	(*═════════════════════════════════════════════════════════*)
	(*  External Systems and I/O    *)
	(*═════════════════════════════════════════════════════════*)
	controlfb_control_b_start                                  , (* BOOL *)
	controlfb_control_b_stop                                   , (* BOOL *)
	controlfb_control_b_shutdown                               , (* BOOL *)
	controlfb_control_b_Reset                                  , (* BOOL *)
	controlfb_control_b_SystemShutdown                         , (* BOOL *)
	controlfb_control_b_EMstop                                 , (* BOOL *)
	controlfb_control_b_ClearHistory                           , (* BOOL *)
	controlfb_control_b_ActivateSettings                       , (* BOOL *)
	controlfb_control_b_startDeHum                             , (* BOOL *)
	controlfb_Operation_inputgrid_b_SyncClose                  , (* BOOL *)
	controlfb_Operation_Genset_b_manualStart                   , (* BOOL *)
	controlfb_Operation_PSB_b_SyncClose                        , (* BOOL *)
	controlfb_Operation_charger_b_StartCharging                , (* BOOL *)
	controlfb_Operation_charger_b_ResetCharger                 , (* BOOL *)
	controlfb_Operation_system_r_NominalVoltage                , (* REAL *)
	controlfb_Operation_system_r_NominalFrequency              , (* REAL *)
	controlfb_Operation_system_r_Pset                          , (* REAL *)
	controlfb_Operation_system_r_Qset                          , (* REAL *)
	controlfb_Operation_system_r_PFset                         , (* REAL *)
	controlfb_Operation_system_b_PFsetEnable                   , (* BOOL *)
	controlfb_Operation_system_b_SounderMute                   , (* BOOL *)
	controlfb_Operation_system_b_SounderTest                   , (* BOOL *)
	controlfb_Operation_system_b_GenGridModeTrans              , (* BOOL *)
	controlfb_Operation_system_b_GridTakeOverEnable            , (* BOOL *)
	controlfb_Operation_parallel_b_DetectSlaves                , (* BOOL *)
	controlfb_Operation_parallel_r_ActivePowerSlave1           , (* REAL *)
	controlfb_Operation_parallel_r_ReactivePowerSlave1         , (* REAL *)
	controlfb_Operation_parallel_r_ActivePowerSlave2           , (* REAL *)
	controlfb_Operation_parallel_r_ReactivePowerSlave2         , (* REAL *)
	controlfb_Operation_BMS_b_ManualStartHVDC                  , (* BOOL *)
	controlfb_SoftSettings_inputgrid_PeakshaveMode             , (* ePeakshaveMode *)
	controlfb_SoftSettings_inputgrid_setpointTimeslot1_r_SocTarget, (* REAL *)
	controlfb_SoftSettings_inputgrid_setpointTimeslot1_r_IdleChargePower, (* REAL *)
	controlfb_SoftSettings_inputgrid_setpointTimeslot1_r_FeedInCurrentLimitSoft, (* REAL *)
	controlfb_SoftSettings_inputgrid_setpointTimeslot1_r_SupplyCurrentLimitSoft, (* REAL *)
	controlfb_SoftSettings_inputgrid_setpointTimeslot2_r_SocTarget, (* REAL *)
	controlfb_SoftSettings_inputgrid_setpointTimeslot2_r_IdleChargePower, (* REAL *)
	controlfb_SoftSettings_inputgrid_setpointTimeslot2_r_FeedInCurrentLimitSoft, (* REAL *)
	controlfb_SoftSettings_inputgrid_setpointTimeslot2_r_SupplyCurrentLimitSoft, (* REAL *)
	controlfb_SoftSettings_inputgrid_b_BreakerControl          , (* BOOL *)
	controlfb_SoftSettings_inputgrid_b_ReverseCTDirection      , (* BOOL *)
	controlfb_SoftSettings_inputgrid_ui_CTrange                , (* UINT *)
	controlfb_SoftSettings_inputgrid_r_VTratio                 , (* REAL *)
	controlfb_SoftSettings_inputgrid_b_GridCodesActive         , (* BOOL *)
	controlfb_SoftSettings_inputgrid_b_WeakGridInput           , (* BOOL *)
	controlfb_SoftSettings_inputgrid_breaker_AutoConnect       , (* BOOL *)
	controlfb_SoftSettings_inputgrid_breaker_ShutdownDisconnect, (* BOOL *)
	controlfb_SoftSettings_inputgrid_breaker_EMstopDisconnect  , (* BOOL *)
	controlfb_SoftSettings_inputgrid_breaker_CurrentLimitDisconnect, (* BOOL *)
	controlfb_SoftSettings_inputgrid_breaker_CurrentLimitRetries, (* BYTE *)
	controlfb_SoftSettings_inputgenset_b_AutoStartStop         , (* BOOL *)
	controlfb_SoftSettings_inputgenset_b_HydridMode            , (* BOOL *)
	controlfb_SoftSettings_inputgenset_b_EnableSchedule        , (* BOOL *)
	controlfb_SoftSettings_inputgenset_setpointTimeslot1_r_SoCStart, (* REAL *)
	controlfb_SoftSettings_inputgenset_setpointTimeslot1_r_SoCStop, (* REAL *)
	controlfb_SoftSettings_inputgenset_setpointTimeslot1_r_BatteryloadStart, (* REAL *)
	controlfb_SoftSettings_inputgenset_setpointTimeslot1_r_BatteryloadStop, (* REAL *)
	controlfb_SoftSettings_inputgenset_setpointTimeslot1_b_StartAtBatteryError, (* BOOL *)
	controlfb_SoftSettings_inputgenset_setpointTimeslot2_r_SoCStart, (* REAL *)
	controlfb_SoftSettings_inputgenset_setpointTimeslot2_r_SoCStop, (* REAL *)
	controlfb_SoftSettings_inputgenset_setpointTimeslot2_r_BatteryloadStart, (* REAL *)
	controlfb_SoftSettings_inputgenset_setpointTimeslot2_r_BatteryloadStop, (* REAL *)
	controlfb_SoftSettings_inputgenset_setpointTimeslot2_b_StartAtBatteryError, (* BOOL *)
	controlfb_SoftSettings_inputgenset_b_PSBExtGensetMonitoring, (* BOOL *)
	controlfb_SoftSettings_inputgenset_b_FreqProtectionEnable  , (* BOOL *)
	controlfb_SoftSettings_inputgenset_Generator_e_GensetMode  , (* eGensetMode *)
	controlfb_SoftSettings_inputgenset_Generator_b_GensetLoadshareLine, (* BOOL *)
	controlfb_SoftSettings_inputgenset_Generator_r_RatedPower  , (* REAL *)
	controlfb_SoftSettings_inputgenset_Generator_r_powerloadMax, (* REAL *)
	controlfb_SoftSettings_inputgenset_Generator_r_PowerloadMin, (* REAL *)
	controlfb_SoftSettings_inputgenset_Generator_r_PowerloadEff, (* REAL *)
	controlfb_SoftSettings_inputgenset_Generator_r_ramprate    , (* REAL *)
	controlfb_SoftSettings_inputgenset_Generator_ui_CooldownTime, (* UINT *)
	controlfb_SoftSettings_inputgenset_Generator_ui_WarmupTime , (* UINT *)
	controlfb_SoftSettings_inputgenset_Loadbank_b_Enable       , (* BOOL *)
	controlfb_SoftSettings_inputgenset_Loadbank_r_PowerRating  , (* REAL *)
	controlfb_SoftSettings_inputgenset_Loadbank_r_PowerStepSize, (* REAL *)
	controlfb_SoftSettings_PSB_PeakshaveMode                   , (* ePeakshaveMode *)
	controlfb_SoftSettings_PSB_setpointTimeslot1_r_SocTarget   , (* REAL *)
	controlfb_SoftSettings_PSB_setpointTimeslot1_r_IdleChargePower, (* REAL *)
	controlfb_SoftSettings_PSB_setpointTimeslot1_r_FeedInCurrentLimitSoft, (* REAL *)
	controlfb_SoftSettings_PSB_setpointTimeslot1_r_SupplyCurrentLimitSoft, (* REAL *)
	controlfb_SoftSettings_PSB_setpointTimeslot2_r_SocTarget   , (* REAL *)
	controlfb_SoftSettings_PSB_setpointTimeslot2_r_IdleChargePower, (* REAL *)
	controlfb_SoftSettings_PSB_setpointTimeslot2_r_FeedInCurrentLimitSoft, (* REAL *)
	controlfb_SoftSettings_PSB_setpointTimeslot2_r_SupplyCurrentLimitSoft, (* REAL *)
	controlfb_SoftSettings_PSB_b_BreakerControl                , (* BOOL *)
	controlfb_SoftSettings_PSB_b_ReverseCTDirection            , (* BOOL *)
	controlfb_SoftSettings_PSB_ui_CTrange                      , (* UINT *)
	controlfb_SoftSettings_PSB_r_VTratio                       , (* REAL *)
	controlfb_SoftSettings_system_b_EnableSchedule             , (* BOOL *)
	controlfb_SoftSettings_system_b_EnableTransportMode        , (* BOOL *)
	controlfb_SoftSettings_system_b_EcoModeEnable              , (* BOOL *)
	controlfb_SoftSettings_system_e_UgridPowerMode             , (* eUgridPowerMode *)
	controlfb_SoftSettings_system_e_NetcontactorMode           , (* eNetcontMode *)
	controlfb_SoftSettings_system_e_UgridPowerLimitingMode     , (* ePLM *)
	controlfb_SoftSettings_system_b_AutomaticSwitching         , (* BOOL *)
	controlfb_SoftSettings_system_b_AMF                        , (* BOOL *)
	controlfb_SoftSettings_system_r_FrequencyDroop             , (* REAL *)
	controlfb_SoftSettings_system_r_VoltageDroop               , (* REAL *)
	controlfb_SoftSettings_system_r_SocMin                     , (* REAL *)
	controlfb_SoftSettings_system_r_SocMax                     , (* REAL *)
	controlfb_SoftSettings_system_r_PDischargeLimit            , (* REAL *)
	controlfb_SoftSettings_system_r_PChargeLimit               , (* REAL *)
	controlfb_SoftSettings_system_r_AMax                       , (* REAL *)
	controlfb_SoftSettings_system_s_SystemName                 , (* STRING(18) *)
	controlfb_SoftSettings_system_s_SMSnumber                  , (* STRING(18) *)
	controlfb_SoftSettings_system_ScheduleTimeSlot1_b_active   , (* BOOL *)
	controlfb_SoftSettings_system_ScheduleTimeSlot1_usi_DayOfWeek, (* USINT *)
	controlfb_SoftSettings_system_ScheduleTimeSlot1_usi_HourOfDay, (* USINT *)
	controlfb_SoftSettings_system_ScheduleTimeSlot1_usi_MinuteOfHour, (* USINT *)
	controlfb_SoftSettings_system_ScheduleTimeSlot2_b_active   , (* BOOL *)
	controlfb_SoftSettings_system_ScheduleTimeSlot2_usi_DayOfWeek, (* USINT *)
	controlfb_SoftSettings_system_ScheduleTimeSlot2_usi_HourOfDay, (* USINT *)
	controlfb_SoftSettings_system_ScheduleTimeSlot2_usi_MinuteOfHour, (* USINT *)
	controlfb_SoftSettings_system_by_LEDbrightness             , (* BYTE *)
	controlfb_SoftSettings_setup_e_AcInputType                 , (* eAcInputType *)
	controlfb_SoftSettings_setup_b_MasterSlaveMode             , (* BOOL *)
	controlfb_SoftSettings_setup_b_PeakshaveBoxEnable          , (* BOOL *)
	controlfb_SoftSettings_setup_e_Gridmode                    , (* eGridmode *)
	controlfb_SoftSettings_setup_e_DcCouplingType              , (* eDCinputType *)
	controlfb_SoftSettings_setup_b_ExtGenset                   , (* BOOL *)
	controlfb_HardSettings_setup_e_ControlSource               , (* eControlSources *)
	controlfb_HardSettings_charger_r_PowerMax                  , (* REAL *)
	controlfb_HardSettings_parallel_b_MasterSlaveEnabled       , (* BOOL *)
	controlfb_HardSettings_parallel_b_UnitIsMaster             , (* BOOL *)
	controlfb_HardSettings_parallel_b_ShutdownOnCommError      , (* BOOL *)
	controlfb_HardSettings_parallel_b_EffiencyMode             , (* BOOL *)
	controlfb_HardSettings_parallel_r_VoltageDroop             , (* REAL *)
	controlfb_HardSettings_parallel_r_FrequencyDroop           , (* REAL *)
	controlfb_HardSettings_system_r_PDischargeLimit            , (* REAL *)
	controlfb_HardSettings_system_r_PChargeLimit               , (* REAL *)
	controlfb_HardSettings_system_r_SMax                       , (* REAL *)
	controlfb_HardSettings_system_r_Amax                       , (* REAL *)
	controlfb_HardSettings_system_e_EarthingSystem             , (* eEarthingSystems *)
	controlfb_HardSettings_system_a_ui_InputCurrentLimit_1     , (* UINT *)
	controlfb_HardSettings_system_a_ui_InputCurrentLimit_2     , (* UINT *)
	controlfb_HardSettings_system_a_ui_OutputCurrentLimit_1    , (* UINT *)
	controlfb_HardSettings_system_a_ui_OutputCurrentLimit_2    , (* UINT *)
	controlfb_HardSettings_system_a_ui_OutputCurrentLimit_3    , (* UINT *)
	Generator_CommunicationOK                                  , (* BOOL *)
	Generator_FuelLow                                          , (* BOOL *)
	Generator_FuelCritical                                     , (* BOOL *)
	Generator_bGenBreakerClosed                                , (* BOOL *)
	Generator_bMainBreakerClosed                               , (* BOOL *)
	Generator_bGenRunning                                      , (* BOOL *)
	Generator_bGenVoltFreqOK                                   , (* BOOL *)
	Generator_bMainsFailure                                    , (* BOOL *)
	Generator_eActiveGenMode                                   , (* eGenOperationMode *)
	Generator_bIslandModeActive                                , (* BOOL *)
	Generator_bAMFActive                                       , (* BOOL *)
	Generator_bPeakshaveActive                                 , (* BOOL *)
	Generator_bFixedPowerActive                                , (* BOOL *)
	Generator_ar_LineVoltage_AVG                               , (* REAL *)
	Generator_ar_LineVoltage_L1                                , (* REAL *)
	Generator_ar_LineVoltage_L2                                , (* REAL *)
	Generator_ar_LineVoltage_L3                                , (* REAL *)
	Generator_ar_PhaseVoltage_AVG                              , (* REAL *)
	Generator_ar_PhaseVoltage_L1                               , (* REAL *)
	Generator_ar_PhaseVoltage_L2                               , (* REAL *)
	Generator_ar_PhaseVoltage_L3                               , (* REAL *)
	Generator_ar_Frequency_AVG                                 , (* REAL *)
	Generator_ar_Frequency_L1                                  , (* REAL *)
	Generator_ar_Frequency_L2                                  , (* REAL *)
	Generator_ar_Frequency_L3                                  , (* REAL *)
	Generator_ar_Current_AVG                                   , (* REAL *)
	Generator_ar_Current_L1                                    , (* REAL *)
	Generator_ar_Current_L2                                    , (* REAL *)
	Generator_ar_Current_L3                                    , (* REAL *)
	Generator_ar_PowerFactor_AVG                               , (* REAL *)
	Generator_ar_ActivePower_AVG                               , (* REAL *)
	Generator_ar_ActivePower_L1                                , (* REAL *)
	Generator_ar_ActivePower_L2                                , (* REAL *)
	Generator_ar_ActivePower_L3                                , (* REAL *)
	Generator_ar_ReactivePower_AVG                             , (* REAL *)
	Generator_ar_ApparentPower_AVG                             , (* REAL *)
	HartingIO_b_DigitalInput1Active                            , (* BOOL *)
	HartingIO_b_DigitalInput2Active                            , (* BOOL *)
	HartingIO_b_GenLowFuel                                     , (* BOOL *)
	HartingIO_b_ExtSystemShutdownRequest                       , (* BOOL *)
	HartingIO_b_ExtEMstopOK                                    , (* BOOL *)
	HartingIO_b_ExtEMstopActive                                , (* BOOL *)
	last
) DINT;
END_TYPE

// ---- POUs/MonitoringControl/IoT/DUTS/eIoTCommVersion.TcDUT
{attribute 'qualified_only'}
{attribute 'strict'}
TYPE eIoTCommVersion :
(
	V1 := 0,
	V2 := 1
);
END_TYPE

// ---- POUs/MonitoringControl/IoT/DUTS/eLogType.TcDUT
{attribute 'qualified_only'}
TYPE eLogType :
(
	none := 0,
	nuc := 1,
	cloud := 2
)UINT;
END_TYPE

// ---- POUs/MonitoringControl/IoT/DUTS/eUpdate.TcDUT
{attribute 'qualified_only'}
TYPE eUpdate :
(
	Fast			:= 0,
	Slow			:= 1,
	OnChange 		:= 2, //Updates only of variable has changed from previous value, but additionaly exactly once at system startup.
	Daily			:= 3
)UINT;
END_TYPE

// ---- POUs/MonitoringControl/IoT/DUTS/e_ORAttributeType.TcDUT
{attribute 'qualified_only'}
{attribute 'strict'}
TYPE e_ORAttributeType :
(
	text := 0,
	number := 2,
	integer := 3,
	JSON := 4
);
END_TYPE

// ---- POUs/MonitoringControl/IoT/DUTS/ST_AutoProvisioning.TcDUT
TYPE ST_AutoProvisioning :
	STRUCT
		sType	: STRING;
		sRealm	: STRING;
		sError	: STRING;
	END_STRUCT
END_TYPE

// ---- POUs/MonitoringControl/IoT/DUTS/ST_IotProps.TcDUT
TYPE ST_IotProps :
STRUCT
	sName		: STRING;
	sValue		: STRING(2000);
	eUpdate 	: eUpdate;
	st_RW		: ST_RW;
	pAdress		: PVOID;
	diSize		: DINT;
	ClassType : __SYSTEM.TYPE_CLASS;
	bNumber		: BOOL;
	bJson		: BOOL;
END_STRUCT
END_TYPE

// ---- POUs/MonitoringControl/IoT/DUTS/ST_RW.TcDUT
TYPE ST_RW :
STRUCT
	ReadFromNUC : BOOL:= FALSE;//enabling Read and Write can create unintended behaviour, consider feedback var
	WriteToNUC: BOOL:=FALSE ; //enabling Read and Write can create unintended behaviour, consider feedback var
END_STRUCT
END_TYPE

// ---- POUs/MonitoringControl/IoT/DUTS/ST_Supervisor.TcDUT
TYPE ST_Supervisor :
	STRUCT
		DATA	: STRING;
		ERROR	: STRING;
	END_STRUCT
END_TYPE

// ---- POUs/MonitoringControl/IoT/DUTS/ST_VarBuffer.TcDUT
TYPE ST_VarBuffer :
STRUCT
	sValue 	  : STRING(2000);
	pAdress   : PVOID;
	diSize	  : DINT;  
	ClassType : __SYSTEM.TYPE_CLASS;
	bNumber   : BOOL;
END_STRUCT
END_TYPE

// ---- POUs/MonitoringControl/IoT/_Structs/ST_IoTDataHMI.TcDUT
TYPE ST_IoTDataHMI :
STRUCT
	Label 				: STRING;
	Varname				: eDataMappingVarNames;
	Unit				: STRING(20);
	LogType 			: eLogType; 
	LogInterval 		: eUpdate;
	b_IOTWriteAllowed	: BOOL;
END_STRUCT
END_TYPE

// ---- POUs/MonitoringControl/IoT/_Structs/ST_IotData_credits.TcDUT
TYPE ST_IotData_credits :
STRUCT
	TotalCredits 		: DINT := 100;
	RemainingCredits	: DINT;
	UsedCredits			: DINT;
END_STRUCT
END_TYPE

// ---- POUs/MonitoringControl/IoT/_Structs/st_IOT_params.TcDUT
TYPE st_IOT_params :
STRUCT
	b_controlEnable			: 	BOOL := FALSE;
	r_UpdateTimeFast		: 	REAL := 15; //seconds
	r_UpdateTimeSlow		: 	REAL := 60; //seconds
	IotCommVersion			: 	eIotCommVersion;
	DefaultLoggingBudget	:	UINT	:= 100;
END_STRUCT
END_TYPE

// ---- POUs/MonitoringControl/IoT/_Structs/ST_IOT_SentStateLog.TcDUT
TYPE ST_IOT_SentStateLog :
STRUCT
	bUpdate			: BOOL;
	bMessageSent	: BOOL;
	LastIndexSent	: INT;
	LastIndex		: INT;
END_STRUCT
END_TYPE

// ---- POUs/MonitoringControl/ProfinetController/enums/eExternalControlMode.TcDUT
{attribute 'qualified_only'}
{attribute 'strict'}
TYPE eExternalControlMode :
(
	off := 0,
	Readonly := 1,
	BasicControl := 2,
	AdvancedControl := 3
);
END_TYPE

// ---- POUs/MonitoringControl/ProfinetController/enums/GenGridMode.TcDUT
{attribute 'qualified_only'}
{attribute 'strict'}
TYPE GenGridMode :
(
	none := 0,
	Grid := 1,
	GridDisconnected := 11,
	GridToNone := 12,
	Genset := 2
);
END_TYPE

// ---- POUs/MonitoringControl/ProfinetController/enums/uSWversion.TcDUT
TYPE uSWversion :
UNION
	a4byte_SWVer 	: 	ARRAY[0..3] OF BYTE;
	UD_SWVer		:	UDINT; 
END_UNION
END_TYPE

// ---- POUs/MonitoringControl/ProfinetController/Structs/future use/ST_PNInput_DCBusExpansion.TcDUT
TYPE ST_PNInput_DCBusExpansion :
STRUCT
	ControlBits	:	DWORD;
END_STRUCT
END_TYPE

// ---- POUs/MonitoringControl/ProfinetController/Structs/future use/ST_PNInput_DCCharger.TcDUT
TYPE ST_PNInput_DCCharger :
STRUCT
	Controlbits	:	DWORD;
	//b_enable?
	//b_resetCharger
	//b_StartCharging
	Powerlimit	:	DWORD;
END_STRUCT
END_TYPE

// ---- POUs/MonitoringControl/ProfinetController/Structs/future use/ST_PNInput_ParallelOperation.TcDUT
TYPE ST_PNInput_ParallelOperation :
STRUCT
	Controlbits			:	DWORD;
	//b_DetectSlaves	
	r_ActivePower		:	DWORD;
	r_reactivePower		:	DWORD;
END_STRUCT
END_TYPE

// ---- POUs/MonitoringControl/ProfinetController/Structs/future use/ST_PNOutput_DCCharger.TcDUT
TYPE ST_PNOutput_DCCharger :
STRUCT
	statusbits		:	DWORD;
	ChargerStatus	:	DWORD;
	ChargePower		:	DWORD;
END_STRUCT
END_TYPE

// ---- POUs/MonitoringControl/ProfinetController/Structs/future use/ST_PNOutput_DCExpansion.TcDUT
TYPE ST_PNOutput_DCExpansion :
STRUCT
	statusbits	: DWORD;
	Busvoltage	: DWORD;
	RatedPower	: DWORD;
	LoadPercentage	: DWORD;
	CurrentPower	: DWORD;
END_STRUCT
END_TYPE

// ---- POUs/MonitoringControl/ProfinetController/Structs/future use/ST_PNOutput_ParallelOperation.TcDUT
TYPE ST_PNOutput_ParallelOperation :
STRUCT
	statusbits		:	DWORD;
	ActivePower		:	DWORD;
	ReactivePower	:	DWORD;
END_STRUCT
END_TYPE

// ---- POUs/MonitoringControl/ProfinetController/Structs/NestedStructs/ST_PNInput_ACDCCharger.TcDUT
TYPE ST_PNInput_ACDCCharger :
STRUCT
	w_Control			:	WORD;
	ui_ACCurrentlimit	:	UINT	:=	0;
	UI_Pset				:	UINT	:=	0;
	ui_SocMaxLimit		:	UINT	:=	100;
	ui_MinGridVoltage	:	Uint	:=	360;
END_STRUCT
END_TYPE

// ---- POUs/MonitoringControl/ProfinetController/Structs/NestedStructs/ST_PNInput_Battery.TcDUT
TYPE ST_PNInput_Battery :
STRUCT
	w_Control		:	WORD;
	ui_SocMinLimit	:	UINT	:=	0;
	ui_SocMaxLimit	:	UINT	:=	100;
END_STRUCT
END_TYPE

// ---- POUs/MonitoringControl/ProfinetController/Structs/NestedStructs/ST_PNInput_GenControl.TcDUT
TYPE ST_PNInput_GenControl :
STRUCT
	w_Control			:	WORD;
	ui_SOCStart			:	UINT;
	ui_SOCStop			:	UINT;
	ui_BattLoadStart	:	UINT;
	ui_BattLoadStop		:	UINT;
	ui_GenPowerMode		:	UINT;
	ui_GenRatedPower	:	UINT;
	ui_GenMaxPowerLevel	:	UINT;
	ui_GenEffPowerLevel	:	UINT;
	ui_GenMinPowerLevel	:	UINT;
	ui_GenWarmupTime	:	UINT;
	ui_GenCooldownTime	:	UINT;
	ui_IsoPowerRamp		:	UINT;
	ui_GeneratorSetpoint : 	UINT;
	ui_StartStopControl	:	uint;	
END_STRUCT
END_TYPE

// ---- POUs/MonitoringControl/ProfinetController/Structs/NestedStructs/ST_PNInput_General.TcDUT
TYPE ST_PNInput_General :
STRUCT
	W_Control				:	WORD;
	ui_HeatBeat				:	UINT;
	ui_GridMode				:	UINT;
	ui_GridFormingSubMode	:	UINT;	
	ui_Earthingsystem		:	UINT;
	GridConnectionMode		:	UINT;
	PrimaryDigOutState		:	UINT := 99;
	SecondaryDigOutState	:	UINT := 99;
	PrimaryDigInState		:	UINT := 99;
	SecondaryDiginState		:	UINT := 99;
END_STRUCT
END_TYPE

// ---- POUs/MonitoringControl/ProfinetController/Structs/NestedStructs/ST_PNInput_InputField.TcDUT
TYPE ST_PNInput_InputField :
STRUCT
	w_Control				:	WORD;
	InputConnectionType		:	UINT;
//	ui_FeedInCurrentLimit	:	UINT;
//	ui_FeedOutCurrentLimit	:	UINT;
//	ui_IdleChargePower 		:	UINT;
//	ui_SocTarget			:	UINT;
//	ui_InputConnectionType	:	UINT;
END_STRUCT                       
END_TYPE

// ---- POUs/MonitoringControl/ProfinetController/Structs/NestedStructs/ST_PNInput_InputGridControl.TcDUT
TYPE ST_PNInput_InputGridControl :
STRUCT
	w_Control				:	WORD;
	ui_FeedInCurrentLimit	:	UINT;
	ui_SupplyCurrentLimit	:	UINT;
	ui_CurrentLimitRetries	:	UINT;
	ui_ContactorControl		:	uint;
END_STRUCT
END_TYPE

// ---- POUs/MonitoringControl/ProfinetController/Structs/NestedStructs/ST_PNInput_PeakShaveBox.TcDUT
TYPE ST_PNInput_PeakShaveBox :
STRUCT
	w_Control			:	WORD;
	ui_FeedInCurrentLimit	:	UINT;
	ui_SupplyCurrentLimit	:	UINT;
	ui_VTRatio				:	UINT;
	UI_CTRatio				:	UINT;
END_STRUCT
END_TYPE

// ---- POUs/MonitoringControl/ProfinetController/Structs/NestedStructs/ST_PNInput_Powerstack.TcDUT
TYPE ST_PNInput_Powerstack :
STRUCT
	w_Control			:	WORD;
	ui_NominalVoltage	:	UINT;
	ui_NominalFrequency	:	UINT;
	i_Pset				:	INT;
	i_Qset				:	INT;
	i_PFset				:	INT;
	ui_FrequencyDroop	:	UINT;
	ui_VoltageDroop		:	UINT;
	ui_PowerRampRate	:	UINT;
	ui_SOCDroopUpshiftStart		:	UINT;
	ui_SOCDroopDownShiftStart	:	UINT;
	ui_PowerLimitMode	:	UINT;
	ui_ACCurrentLimit	:	UINT;
END_STRUCT
END_TYPE

// ---- POUs/MonitoringControl/ProfinetController/Structs/NestedStructs/ST_PNOutput_ACDCCharger.TcDUT
TYPE ST_PNOutput_ACDCCharger :
STRUCT
	w_Status						: WORD;
	w_Warnings						: WORD;
	w_Faults						: WORD;
	ui_ChargerStatus				: WORD;
	TotalChargerPower				: WORD;
	AvailableChargePower			: UINT;
	ActivePower						: UINT;
	Frequency						: UINT;
	VoltageAB						: UINT;
	VoltageBC						: UINT;
	VoltageCA						: UINT;
	CurrentL1						: UINT;
	CurrentL2						: UINT;
	CurrentL3						: UINT;
	ui_ACCurrentLimitAct			: UINT;
	ui_PSetAct						: UINT;
	ui_SocLimitAct					: UINT;
	ui_MinGridVoltageAct			: UINT;
END_STRUCT
END_TYPE

// ---- POUs/MonitoringControl/ProfinetController/Structs/NestedStructs/ST_PNOutput_Battery.TcDUT
TYPE ST_PNOutput_Battery :
STRUCT
	ui_Status						: UINT;
	w_Warnings						: WORD;
	w_Faults						: WORD;

	ui_SOC							: UINT;
	ui_SOH							: UINT;
	ui_DClinkVoltage 				: UINT;
	i_DClinkCurrent 				: INT;
	ui_MaxAllowedDischargeCurrent 	: UINT;
	ui_MaxAllowedChargeCurrent 		: UINT;
	i_MinCellTemperature 			: INT;
	i_MaxCellTemperature			: INT;
	ui_RemainingChargeEnergy 		: UINT;
	ui_RemainingDischargeEnergy 	: UINT;
	ui_CycleCount					: UINT;
END_STRUCT
END_TYPE

// ---- POUs/MonitoringControl/ProfinetController/Structs/NestedStructs/ST_PNOutput_GenControl.TcDUT
TYPE ST_PNOutput_GenControl :
STRUCT
	w_Status					:	WORD;
	w_Warnings					:	WORD;
	w_Faults					:	WORD;
	ui_GeneratorStatus			:	UINT;	
END_STRUCT
END_TYPE

// ---- POUs/MonitoringControl/ProfinetController/Structs/NestedStructs/ST_PNOutput_General.TcDUT
TYPE ST_PNOutput_General :
STRUCT
	ui_SystemState				:	UINT;
	w_SystemStatus				:	WORD;	
	w_SystemWarnings			:	WORD;
	w_SystemFaults				:	WORD;
	w_CoolingSystemStatus		:	WORD;
	w_CoolingSystemWarnings		:	WORD;
	w_CoolingSystemFaults		:	WORD;
	w_InternalSupplyStatus		:	WORD;
	w_InternalSupplyWarnings	:	WORD;
	w_InternalSupplyFaults		:	WORD;	
	ui_HeartBeatOut				:	UINT;
	ui_Gridmode					: 	UINT;
	ui_GridFormingSubMode		: 	UINT;
	udi_SerialNumber			:	UDINT;
	dw_SWVersion				:	DWORD;
	//ui_InputConnectionType		:	UINT;
END_STRUCT
END_TYPE

// ---- POUs/MonitoringControl/ProfinetController/Structs/NestedStructs/ST_PNOutput_InputField.TcDUT
TYPE ST_PNOutput_InputField:
STRUCT
	w_Status					:	WORD;
	w_Warnings					:	WORD;
	w_Faults					:	WORD;
	ui_InputConnectionType		:	UINT;
	ui_InputConnectionState		:	UINT;
	i_ActivePower				:	INT;
	i_ReactivePower				:	INT;
	i_PowerFactor				:	INT;
	ui_Frequency				:	UINT;
	ui_VoltageL1N				:	UINT;
	ui_VoltageL2N				:	UINT;
	ui_VoltageL3N				:	UINT;
	ui_VoltageL1L2				:	UINT;
	ui_VoltageL2L3				:	UINT;
	ui_VoltageL3L1				:	UINT;
	ui_CurrentL1				:	UINT;
	ui_CurrentL2				:	UINT;
	ui_CurrentL3				:	UINT;
	ui_CurrentN					:	UINT;
	ui_CurrentLimitField		:	UINT;
	udi_TotalEnergySupplied 	:	UDINT;
	udi_TotalEnergyConsumed 	:	UDINT;
	ui_Current1L1				:	UINT;
	ui_Current1L2				:	UINT;
	ui_Current1L3				:	UINT;
	ui_Current1N				:	UINT;
	ui_Current2L1				:	UINT;
	ui_Current2L2				:	UINT;
	ui_Current2L3				:	UINT;
	ui_Current2N				:	UINT;
END_STRUCT
END_TYPE

// ---- POUs/MonitoringControl/ProfinetController/Structs/NestedStructs/ST_PNOutput_InputGridControl.TcDUT
TYPE ST_PNOutput_InputGridControl :
STRUCT
	w_Status					:	WORD;
	w_Warnings					:	WORD;
	w_Faults					:	WORD;
	ui_InputGridStatus			:	UINT;
END_STRUCT
END_TYPE

// ---- POUs/MonitoringControl/ProfinetController/Structs/NestedStructs/ST_PNOutput_OutputField.TcDUT
TYPE ST_PNOutput_OutputField:
STRUCT
	w_Status					:	WORD;
	w_Warnings					:	WORD;
	w_Faults					:	WORD;
	i_ActivePower				:	INT;
	i_ReactivePower				:	INT;
	i_PowerFactor				:	INT;
	ui_Frequency				:	UINT;
	ui_VoltageL1N				:	UINT;
	ui_VoltageL2N				:	UINT;
	ui_VoltageL3N				:	UINT;
	ui_VoltageL1L2				:	UINT;
	ui_VoltageL2L3				:	UINT;
	ui_VoltageL3L1				:	UINT;
	ui_CurrentL1				:	UINT;
	ui_CurrentL2				:	UINT;
	ui_CurrentL3				:	UINT;
	ui_CurrentN					:	UINT;
	ui_CurrentLimitField		:	UINT;
	udi_TotalEnergySupplied 	:	UDINT;
	udi_TotalEnergyConsumed 	:	UDINT;
	ui_Current1L1				:	UINT;
	ui_Current1L2				:	UINT;
	ui_Current1L3				:	UINT;
	ui_Current1N				:	UINT;
	ui_Current2L1				:	UINT;
	ui_Current2L2				:	UINT;
	ui_Current2L3				:	UINT;
	ui_Current2N				:	UINT;
	ui_Current3L1				:	UINT;
	ui_Current3L2				:	UINT;
	ui_Current3L3				:	UINT;
	ui_Current3N				:	UINT;
END_STRUCT
END_TYPE

// ---- POUs/MonitoringControl/ProfinetController/Structs/NestedStructs/ST_PNOutput_PeakShaveBox.TcDUT
TYPE ST_PNOutput_PeakShaveBox:
STRUCT
	w_Status					:	WORD;
	w_Warnings					:	WORD;
	w_Faults					:	WORD;
	i_ActivePower				:	INT;
	i_ReactivePower				:	INT;
	i_PowerFactor				:	INT;
	ui_Frequency				:	UINT;
	ui_VoltageL1N				:	UINT;
	ui_VoltageL2N				:	UINT;
	ui_VoltageL3N				:	UINT;
	ui_VoltageL1L2				:	UINT;
	ui_VoltageL2L3				:	UINT;
	ui_VoltageL3L1				:	UINT;
	ui_CurrentL1				:	UINT;
	ui_CurrentL2				:	UINT;
	ui_CurrentL3				:	UINT;
	ui_CurrentN					:	UINT;
END_STRUCT
END_TYPE

// ---- POUs/MonitoringControl/ProfinetController/Structs/NestedStructs/ST_PNOutput_PowerStack.TcDUT
TYPE ST_PNOutput_PowerStack :
STRUCT
	w_Status					:	WORD;
	w_Warnings					:	WORD;
	w_Faults					:	WORD;
	
	ui_PowerStackStatus			: UINT;
	i_ActivePower				: INT;
	i_ReactivePower				: INT;
	ui_SupplyVoltage			: UINT;
	ui_Supplyfrequency			: UINT;
	ui_ACCurrent				: UINT;
	i_PsetAct					: INT;
	i_QsetAct					: INT;
	i_PFSetAct					: UINT;
	ui_LoadPercentage			: UINT;
	ui_RatedCurrent				: UINT;
	ui_RatedPower				: UINT;
	ui_DischargePowerLimit		: UINT;
	ui_ChargePowerLimit			: UINT;
	ui_ACcurrentLimit			: UINT;
	ui_ApparentPowerLimit		: UINT;
	ui_ReactivePowerLimit		: UINT;
END_STRUCT
END_TYPE

// ---- POUs/MonitoringControl/ProfinetController/Structs/NestedStructs/ST_PNOutput_ZPT.TcDUT
TYPE ST_PNOutput_ZPT :
STRUCT
	w_Status					:	WORD;
	w_Warnings					:	WORD;
	w_Errors					:	WORD;
	ui_RatedPower				:	UINT;
	ui_Powerload				:	UINT;
	i_TransformerTemperature	:	INT;
END_STRUCT
END_TYPE

// ---- POUs/MonitoringControl/ProfinetController/Structs/ST_PNcontroller_params.TcDUT
TYPE ST_PNcontroller_params :
STRUCT
	b_BigEndian				: BOOL;
	b_testComm				: BOOL;
	b_MonitoringEnable		: BOOL := TRUE;
	b_ControlEnable			: BOOL := TRUE;
	w_CommTimeOut			: WORD := 10000; // milli seconds
	TestVars				: ST_PNTest;
	Limits					: ST_ExtController_limits;
END_STRUCT
END_TYPE

// ---- POUs/MonitoringControl/ProfinetController/Structs/ST_PNinput.TcDUT
TYPE ST_PNinput :
STRUCT
	PNIOBoxState		:	WORD;
	PNIOBoxDiag			:	WORD;	
	General 			: ST_PNInput_General;
	Battery				: ST_PNInput_Battery;
	Inputfield			: ST_PNInput_InputField;
	PSB					: ST_PNInput_PeakshaveBox;
	Powerstack			: ST_PNInput_Powerstack;
	GenControl 			: ST_PNInput_GenControl;
	InputGridControl	: ST_PNInput_InputGridControl;	
	ACDCCharger			: ST_PNInput_ACDCCharger;
END_STRUCT
END_TYPE

// ---- POUs/MonitoringControl/ProfinetController/Structs/ST_PNOutput.TcDUT
TYPE ST_PNOutput :
STRUCT
	General 		: ST_PNOutput_General;
	Battery			: ST_PNOutput_Battery;
	OutputField		: ST_PNOutput_Outputfield;
	InputField		: ST_PNOutput_Inputfield;
	Powerstack 		: ST_PNOutput_Powerstack;
	PSB 			: ST_PNOutput_PeakshaveBox;
	ZPT				: ST_PNOutput_ZPT;
	GenControl 		: ST_PNOutput_GenControl;
	InputGridControl: ST_PNOutput_InputGridControl;
	ACDCCharger		: ST_PNOutput_ACDCCharger;
END_STRUCT
END_TYPE

// ---- POUs/MonitoringControl/ProfinetController/Structs/ST_PNTest.TcDUT
TYPE ST_PNTest :
STRUCT
	b_CheckMonitoring	: BOOL;
	b_MonitoringOK		: BOOL;
	s_MonitoringErr		: STRING;
	i_Pset				: INT;
	i_Qset				: INT;
	w_SetAddress		: WORD;
	w_SetValue			: WORD;
	bit_start			: BOOL;
	bit_stop			: BOOL;
	bit_Shutdown		: BOOL;
	bit_SystemShutdown	: BOOL;
	bit_Reset			: BOOL;
	bit_EMStop			: BOOL;
	bit_AdvancedControl	: BOOL;
	bit_AutoSwitching	: BOOL;
	bit_Transportmode	: BOOL;
END_STRUCT
END_TYPE

// ---- POUs/MonitoringControl/_Enums/eAcInputType.TcDUT
{attribute 'qualified_only'}
{attribute 'strict'}
TYPE eAcInputType :
(
	None 	:= 0,
	Grid 	:= 1,
	Genset	:= 2
);
END_TYPE

// ---- POUs/MonitoringControl/_Enums/eCapTestSTate.TcDUT
{attribute 'qualified_only'}
{attribute 'strict'}
TYPE eCapTestSTate :
(
	init 				:= 	0,
	WriteSerial			:=	1,
	WriteNameplateCap	:=	2,
	WriteDatetime		:=	3,
	StartSystem 		:= 	4,
	InitialCharge 		:= 	5,
	RestPeriod1			:= 	6,
	DischargeCycle 		:= 	7,
	RestPeriod2 		:= 	8,
	ChargeCycle 		:= 	9,
	RestPeriod3 		:= 	10,
	StopSystem  		:= 	11,
	done				:=	12
);
END_TYPE

// ---- POUs/MonitoringControl/_Enums/eControlSources.TcDUT
{attribute 'qualified_only'}
{attribute 'strict'}
{attribute 'to_string'}
TYPE eControlSources :
(
	Local 				:= 0,
	ExternalController 	:= 1,
	PowerNet			:= 2	
);
END_TYPE

// ---- POUs/MonitoringControl/_Enums/eDcInputType.TcDUT
{attribute 'qualified_only'}
{attribute 'strict'}
TYPE eDcInputType :
(
	None := 0,
	Dc_charger := 1, 
	Dc_extender := 2
);
END_TYPE

// ---- POUs/MonitoringControl/_Enums/eEarthingSystems.TcDUT
{attribute 'qualified_only'}
{attribute 'strict'}
TYPE eEarthingSystems :
(
	None 		:= 0,	
	TN			:= 1,
	TN_ext		:= 2,
	IT			:= 3		
);
END_TYPE

// ---- POUs/MonitoringControl/_Enums/eGridFormingMode.TcDUT
{attribute 'qualified_only'}
{attribute 'strict'}
TYPE eGridFormingMode:
(
	Island := 0,
	Droop := 1
);
END_TYPE

// ---- POUs/MonitoringControl/_Enums/eGridMode.TcDUT
{attribute 'qualified_only'}
{attribute 'strict'}
{attribute 'to_string'}
TYPE eGridMode :
(
	auto := 0,
	following := 1,
	forming	:= 2
);
END_TYPE

// ---- POUs/MonitoringControl/_Enums/eNetContactorDirection.TcDUT
{attribute 'qualified_only'}
{attribute 'strict'}
TYPE eNetContactorDirection :
(
	Left 	:= -1,
	None 	:= 0,
	Right 	:= 1
);
END_TYPE

// ---- POUs/MonitoringControl/_Enums/eOperationMode.TcDUT
{attribute 'qualified_only'}
{attribute 'strict'}
TYPE eOperationMode :
(
	Auto := 0,
	Gridfollowing := 1,
	GridForming	:= 2
);
END_TYPE

// ---- POUs/MonitoringControl/_Enums/ePeakshaveMode.TcDUT
{attribute 'qualified_only'}
{attribute 'strict'}
TYPE ePeakshaveMode :
(
	Multiphase := 0,
	Singlephase := 1
);
END_TYPE

// ---- POUs/MonitoringControl/_Enums/eSchedulerMode.TcDUT
{attribute 'qualified_only'}
{attribute 'strict'}
TYPE eSchedulerMode :
(
	continous := 0,
	daily := 1,
	weekly := 2
);
END_TYPE

// ---- POUs/MonitoringControl/_Enums/ePowerControlType.TcDUT
{attribute 'qualified_only'}
{attribute 'strict'}
{attribue 'to_string}
TYPE ePowerControlType :
(
	Current := 0,
	Power	:=1,
	Both	:= 2
);
END_TYPE

// ---- POUs/MonitoringControl/_Enums/eSystemState.TcDUT
{attribute 'qualified_only'}
{attribute 'strict'}
{attribute 'to_string'}
TYPE eSystemState :
(
	Off 			:= 0,
	Shutdown 		:= 1,
	StandBy 		:= 2,
	Conditioning 	:= 3,
	Starting		:= 4,
	Running			:= 5,
	Charging_Only	:= 6,
	Discharging_Only:= 7,
	Stopped			:= 8,
	EMstop			:= 9,
	Reset			:= 10,
	Init			:= 11,
	Transport		:= 12,
	Dehumidifying	:= 13
);
END_TYPE

// ---- POUs/MonitoringControl/_Enums/eUgridPowerMode.TcDUT
{attribute 'qualified_only'}
{attribute 'strict'}
{attribute 'to_string'}
TYPE eUgridPowerMode :
(
	auto 			:= 0,
	DroopZeroStart	:= 1,
	Droop			:= 2,
	Isochronous		:= 3,
	None			:= 4
);
END_TYPE

// ---- POUs/MonitoringControl/_Structs/ST_ExtController_Events.TcDUT
TYPE ST_ExtController_Events :
STRUCT
	b_HeartbeatFault			: BIT;
	b_couplerError				:	bit;
	
	// control limit warnings
	b_FeedInLimitOutOfRange		: BIT;
	b_SupplyLimitOutOfRange 	: BIT;
	b_IdleChargePowerOutofRange	: BIT;
	b_BatOloadStartOutOfRange	: BIT;
	b_BatOloadStopOutOfRange	: BIT;
	b_SocTargetOutOfRange		: BIT;
	b_SocStartOutOfRange		: BIT;
	b_SocStopOutOfRange			: BIT;
	b_PsetOutOfRange			: BIT;
	b_QsetOutOfRange			: BIT;
	b_PFsetOutOfRange			: BIT;
	b_NominalVoltageOutOfRange	: BIT;
	b_NominalFreqOutOfRange		: BIT;
	b_FreqDroopOutOfRange		: BIT;
	b_VoltageDroopOutOfRange	: BIT;
	b_PmaxOutOfRange			: BIT;
	b_PminOutOfRange			: BIT;
	b_SmaxOutOfRange			: BIT;
	b_AmaxOutOfRange			: BIT;
	b_PowerRamprateOutOfRange	: BIT;
	b_PSBFeedInLimitOutOfRange	: BIT;
	b_PSBSupplyLimitOutOfRange: BIT;
	b_PSBIdleChargePowerOutOfRange: BIT;
	b_PSBSoCTargetOutOfRange	: BIT;
	b_SoCHighLimitOutOfRange	: BIT;
	b_SoCLowLimitOutOfRange		: BIT;
	b_GridModeValueOutOfRange	: BIT;
	b_PowermodeValueOutOfRange	: BIT;

END_STRUCT
END_TYPE

// ---- POUs/MonitoringControl/_Structs/ST_ExtController_get.TcDUT
TYPE ST_ExtController_get :
STRUCT
	control							: ST_ControlVars;
	Operation						: ST_OperationVars;
	SoftSettings					: ST_SoftSettings;
	HardSettings					: ST_HardSettings;
	events							: ST_ExtController_Events;
	b_AdvancedControl				: BOOL;
	ui_Heartbeat					: UINT;
	s_dashboardID					: STRING;
	b_Active						: BOOL;
	e_ConnectionState				: eConnectionState;
	s_OutputJson					: STRING(2000);
	LoggingBudgetOK					: BOOL := TRUE;
END_STRUCT
END_TYPE

// ---- POUs/MonitoringControl/_Structs/ST_ExtController_limits.TcDUT
TYPE ST_ExtController_limits :
STRUCT
	r_InputCtLimit			: REAL := 800;
	r_InverterPowerLimit	: REAL := 360;
	r_InverterCurrentLimit	: REAL := 520;
	r_NominalVoltageMin		: REAL := 360;
	r_NominalVoltageMax		: REAL := 440;
	r_NominalFreqMin		: REAL := 47.5;
	r_NominalFreqMax		: REAL := 52.5;
	r_DroopMax				: REAL := 10; 
	r_PowerRampLimit		: REAL := 300; //%/s
	r_PSBCtLimit			: REAL := 4000;
END_STRUCT
END_TYPE

// ---- POUs/MonitoringControl/_Structs/ST_ExtController_Set.TcDUT
TYPE ST_ExtController_Set :
STRUCT
	b_available				: BOOL;
END_STRUCT
END_TYPE

// ---- POUs/MonitoringControl/_Structs/ST_PLCPersistentVars.TcDUT
TYPE ST_PLCPersistentVars :
STRUCT
	Hardsettings					: ST_HardSettings; 
	Softsettings					: ST_Softsettings;
END_STRUCT
END_TYPE

// ---- POUs/Objects/4Grouter/Struct/dwtoreal.TcDUT
TYPE dwtoreal :
UNION
	Registers	:	ARRAY[1..2] OF WORD;
	dwordvalue	:	dword;
	realvalue	:	REAL;
END_UNION
END_TYPE

// ---- POUs/Objects/4Grouter/Struct/eModemState.TcDUT
{attribute 'qualified_only'}
//{attribute 'strict'}
TYPE eModemState :
(
	Disconnected := 0,
	Connected := 1
);
END_TYPE

// ---- POUs/Objects/4Grouter/Struct/eNetworkState.TcDUT
{attribute 'qualified_only'}
//{attribute 'strict'}
TYPE eNetworkState :
(
	unknown := 0,
	searching := 1,
	Unregistered := 2,
	Registered := 3,
	Roaming := 4
	);
END_TYPE

// ---- POUs/Objects/4Grouter/Struct/eSimSelectionMode.TcDUT
{attribute 'qualified_only'}
{attribute 'strict'}
TYPE eSimSelectionMode :
(
	auto := 0,
	force_sim1 := 1,
	force_sim2 := 2
);
END_TYPE

// ---- POUs/Objects/4Grouter/Struct/eSimState.TcDUT
{attribute 'qualified_only'}
//{attribute 'strict'}
TYPE eSimState :
(
	no_sim := 0,
	Inserted := 1,
	active := 2,
	pin_fault := 3
);
END_TYPE

// ---- POUs/Objects/4Grouter/Struct/eSMSStatus.TcDUT
{attribute 'qualified_only'}
//{attribute 'strict'}
TYPE eSMSStatus :
(
	Idle 			:= 	0,
	NewMessage 		:= 	1,
	SendingMessage 	:= 	2,
	error			:=	3
);
END_TYPE

// ---- POUs/Objects/4Grouter/Struct/eWifiSecurityTypes.TcDUT
{attribute 'qualified_only'}
{attribute 'strict'}
{attribute 'to_string'}
TYPE eWifiSecurityTypes :
(
	none := 0,
	PSK2 := 1,
	SAE  := 2,
	SAE_mixed := 3,
	PSK := 4	
);
END_TYPE

// ---- POUs/Objects/4Grouter/Struct/eWifiStatus.TcDUT
{attribute 'qualified_only'}
TYPE eWifiStatus :
(
	invalid := 0,
	off := 1,
	searching := 2,
	Connected := 3,
	Starting := 4,
	Active := 5
);
END_TYPE

// ---- POUs/Objects/4Grouter/Struct/st_Device.TcDUT
TYPE st_Device :
STRUCT
	SystemUptime	:	UDINT;	
	Temperature		:	REAL;
	RouterSerial	:	STRING(32);
END_STRUCT
END_TYPE

// ---- POUs/Objects/4Grouter/Struct/st_GPS.TcDUT
TYPE st_GPS :
STRUCT
	Latitude 	: 	REAL;
	Longitude 	: 	REAL;
	FixTime 	: 	STRING(32);
	DateTime	:	DT;
	Speed		:	REAL;
	SatCount	:	UINT;
	Accuracy	:	REAL;	
END_STRUCT
END_TYPE

// ---- POUs/Objects/4Grouter/Struct/st_mobile.TcDUT
TYPE st_mobile :
STRUCT
	NetworkOperator				:	STRING(32);
	NetworkInfo					:	STRING(32);
	NetworkType					:	STRING(32);
	RSSI						:	DINT;
	ui_Sim1DataSendMonth		:	UINT;
	ui_Sim1DataReceivedMonth	:	UINT;
	ui_Sim2DataSendMonth		:	UINT;
	ui_Sim2DataReceivedMonth	:	UINT;
	s_EmergencySMSNumber		:	STRING(20);
	s_SecondarySMSNumber		:	STRING(20);
	s_EmergencySMSDevName		:	STRING(18);
	st_LatestSMSMessage			:	STRING(80);
	ModemState					:	eModemState;
	NetworkState				:	eNetworkState;
	ui_ActiveSim				:	UINT;
	SimStatus					:	eSimState;
END_STRUCT
END_TYPE

// ---- POUs/Objects/4Grouter/Struct/st_router_get.TcDUT
TYPE st_router_get :
STRUCT
	Device 		: 	st_Device;
	GPS			:	st_GPS;
	Mobile		:	st_mobile;
	Wifi		:	st_Wifi;
	e_SMSStatus : 	eSMSStatus;
	Events		:	st_Router_Events;
END_STRUCT
END_TYPE

// ---- POUs/Objects/4Grouter/Struct/ST_Router_params.TcDUT
TYPE ST_Router_params :
STRUCT
	IP_TELTONIKA		: STRING(16) := '192.168.1.1';
	MBPort_TELTONIKA 	: UINT := 502;
	T_MBTimeout			: TIME := T#2S;
	MinimumPhoneNumberLength	:UINT := 10;
	
	//temporary setup via stparams until integrated into HMI
	ManualSettings		:	st_router_set;
END_STRUCT
END_TYPE

// ---- POUs/Objects/4Grouter/Struct/st_Router_Events.TcDUT
TYPE st_Router_Events :
STRUCT
	b_MBCommWarning		:	BOOL;
	b_NoSimWarning		:	BOOL;
	b_NoNetworkWarning	: 	BOOL;
	b_noGPSFixWarning	:	BOOL;
	b_SMSNotSendError	:	BOOL; 
	b_NoSMSNumberAvailable	:	BOOL;
	b_TimeUpdateFailed 	: BOOL;
END_STRUCT
END_TYPE

// ---- POUs/Objects/4Grouter/Struct/ST_Router_set.TcDUT
TYPE ST_Router_set :
STRUCT
	EnableWifiClient	:	BOOL;
	WifiClientSSID		:	STRING(32) := 'MachineAccessPoint@VDL';
	WifiClientPass		:	STRING(32) := 'e4ff1c12kLL';
	WifiClientSecType	:	eWifiSecurityTypes := eWifiSecurityTypes.PSK2;
	
	EnableWifiAP		:	BOOL;
	WifiAPSSID			:	STRING(32) := 'ePU10_AP';
	WifiAPPass			:	STRING(32) := 'Welkom!VDL';
	WifiAPSecType		:	eWifiSecurityTypes := eWifiSecurityTypes.PSK2;
	
	SimSelectionMode	:	eSimSelectionMode := eSimSelectionMode.auto;
	Sim1Pin				:	STRING(4) := '0000';
	Sim2Pin				:	STRING(4) := '0000';
	
	UpdateSystemTime	:	BOOL;
	
	AutoRebootEnable	:	BOOL;
	ManualReboot		:	BOOL;
END_STRUCT
END_TYPE

// ---- POUs/Objects/4Grouter/Struct/st_Wifi.TcDUT
TYPE st_Wifi :
STRUCT
	WifiClienModeStatus		:	eWifiStatus;
	WifiAPModeStatus		:	eWifiStatus;
	WifiApNumberOfClients	:	Uint;
END_STRUCT
END_TYPE

// ---- POUs/Objects/ACDCCharger/Enums/eAcDcChargerState.TcDUT
{attribute 'qualified_only'}
{attribute 'strict'}
{attribute 'to_string'} 

TYPE eAcDcChargerState :
(
	init 		:= 0,
	off 		:= 1,
	Standby	 	:= 2,
	starting 	:= 4,
	running		:=	5,
	stopping	:=	6, 

	fault 		:= 7
);
END_TYPE

// ---- POUs/Objects/ACDCCharger/Structs/Hadi/E_ChargerState.TcDUT
TYPE E_ChargerState :
(
    Idle := 0,
    ModulesOff := 10,
    SetVI := 20,
    CheckVoltage := 30,
    EnableModules := 40,
    Running := 100,
    Shutdown := 200,
    OpenRelay := 210,
    Fault := 900
);
END_TYPE

// ---- POUs/Objects/ACDCCharger/Structs/Hadi/ST_CanId.TcDUT
TYPE ST_CanId :
STRUCT
    ExtendedBit : BOOL;   // Bit31 (should always be TRUE)
    ErrorCode   : BYTE;   // Bits 28..26
    DeviceNo    : BYTE;   // Bits 25..22
    CommandNo   : BYTE;   // Bits 21..16
    TargetAddr  : BYTE;   // Bits 15..8
    SourceAddr  : BYTE;   // Bits 7..0
END_STRUCT
END_TYPE

// ---- POUs/Objects/ACDCCharger/Structs/Hadi/ST_ChargerControl.TcDUT
TYPE ST_ChargerControl :
STRUCT
    (* Charger control *)
    bStartCharge      : BOOL;   // start charging sequence
    bStopCharge       : BOOL;   // stop charging sequence

    (* Module enable command *)
    bEnableModules    : BOOL;   // CMD 1A

    (* Setpoints *)
    rSetVoltage       : REAL;   // desired voltage [V]
    rSetCurrent       : REAL;   // desired current [A]

    (* Apply commands *)
    bApplyGroupSet    : BOOL;   // CMD 1B (group control)
    bApplyModuleSet   : BOOL;   // CMD 1C (module control)

    (* Target module *)
    ModuleTarget      : BYTE;   // module number (peer-to-peer)

    (* Hardware relay *)
    bSystemRelayCmd   : BOOL;   // command to close system relay
END_STRUCT
END_TYPE

// ---- POUs/Objects/ACDCCharger/Structs/Hadi/ST_Control.TcDUT
TYPE ST_Control :
STRUCT
	rLimitInputCurrent	: REAL;	// CMD 0F Limit input current on all power modules
//	stModuleControl		: ARRAY [0..10] OF REAL;
	bEnableDisable		: BOOL; // CMD 1A (Broadcastong or Group)
	rSetOutputVoltage	: REAL;	// CMD 1B
	rSetOutputCurrent	: REAL;	// CMD 1B
	bResetMode			: BOOL;	// CMD 1E
	
END_STRUCT
END_TYPE

// ---- POUs/Objects/ACDCCharger/Structs/Hadi/ST_Data.TcDUT
TYPE ST_Data :
STRUCT
	rSystemOutVoltageDc		: REAL;		// CMD 01
	rSystemOutCurrentDc		: REAL;		// CMD 01
	rNumberOfModules		: REAL;		// CMD 02
	stModuleData			: ARRAY [0..10] OF ST_ModuleData;
	
	
	
	
	
END_STRUCT
END_TYPE

// ---- POUs/Objects/ACDCCharger/Structs/Hadi/ST_ModuleControl.TcDUT
TYPE ST_ModuleControl :
STRUCT
	bEnableDisable		: BOOL; // CMD 1A
	rSetOutputVoltage	: REAL;	// CMD 1C
	rSetOutputCurrent	: REAL;	// CMD 1C
	
	
	
	
END_STRUCT
END_TYPE

// ---- POUs/Objects/ACDCCharger/Structs/Hadi/ST_ModuleData.TcDUT
TYPE ST_ModuleData :
STRUCT
	rOutVoltageDc		: REAL;	// CMD 03
	rOutCurrentDc		: REAL;	// CMD 03
	rTemprature			: REAL;	// CMD 04
	rStatus0			: REAL;	// CMD 04
	rStatus1			: REAL;	// CMD 04
	rStatus2			: REAL;	// CMD 04
	rVoltageL1L2		: REAL;	// CMD 06
	rVoltageL2L3		: REAL;	// CMD 06
	rVoltageL3L1		: REAL;	// CMD 06
	rExternalVoltageDc	: REAL;	// CMD 0C      this could be the same as rOutVoltageDc CMD 03
	ravilableCurrentDc	: REAL;	// CMD 0C
	
	 stStatus           : ST_ModuleStatus;  // decoded status bits
	 
	 bValid		: BOOL; // validate if data are updating
	
END_STRUCT
END_TYPE

// ---- POUs/Objects/ACDCCharger/Structs/Hadi/ST_ModuleStatus.TcDUT
TYPE ST_ModuleStatus :
STRUCT
	 (* STATUS 2 *)
    bPfcOff              : BOOL;	// Bit 7
    bInputOverVoltage    : BOOL;	// Bit 6	
    bInputUnderVoltage   : BOOL;	// Bit 5
    bInputAsymmetry      : BOOL;	// Bit 4
    bPhaseLost           : BOOL;	// Bit 3
    bLoadSharingError    : BOOL;	// Bit 2
    bModuleIdDuplicate   : BOOL;	// Bit 1
    bPowerLimitation     : BOOL;	// Bit 0

    (* STATUS 1 *)
    bCanTimeout          : BOOL;	// Bit 7    /////////
    bSlowStartup         : BOOL;	// Bit 6
    bOutputOverVoltage   : BOOL;	// Bit 5
    bTempHigh            : BOOL;	// Bit 4
    bFanError            : BOOL;	// Bit 3
    bModuleProtection    : BOOL;	// Bit 2
    bModuleError         : BOOL;	// Bit 1      ////////////
    bDcSideOff           : BOOL;	// Bit 0

    (* STATUS 0 *)
    bDischargeAbnormal   : BOOL;	// Bit 5
    bMpptSwitchMode      : BOOL;	// Bit 4
    bPfcAbnormal         : BOOL;	// Bit 3
    bInternalCommError   : BOOL;	// Bit 2
    bOutputShortCircuit  : BOOL;	// Bit 0
END_STRUCT
END_TYPE

// ---- POUs/Objects/ACDCCharger/Structs/ST_ACDCCharger_events.TcDUT
TYPE ST_ACDCCharger_events :
STRUCT
	b_CommunicationFault			:	BOOL;
	b_BuscouplerNotFound			:	BOOL;
	b_ACUnderVoltageDeratingActive	: 	BOOL;
	b_BatteryLimitDeratingActive	:	BOOL;
	b_TemperatureDeratingActive		:	BOOL;
	b_CurrentLimitActive			:	BOOL;
	b_SOCLimitReached				:	BOOL;
	b_FailedToGenerateDCOutput		:	BOOL;
	B_ACPhaselossFault				:	BOOL;
	B_ACUndervoltage				:	BOOL;
	B_ACOvervoltage					:	BOOL;
END_STRUCT
END_TYPE

// ---- POUs/Objects/ACDCCharger/Structs/ST_ACDCCharger_get.TcDUT
TYPE ST_ACDCCharger_get :
STRUCT
	e_SystemStatus			: eAcDCChargerState := eACDCChargerState.init;
	
	by_NoModulesActive		: BYTE;	
	by_NoModulesInstalled	: BYTE;
	e_ChargerStatus 		: ARRAY [0..6] OF eAcDcChargerState;
	
	ar_ACvoltage			: ARRAY [0..3] OF REAL;
	r_AvailablePower		: REAL;
	ACmeasurements			: ST_MeasurementFieldData;
	r_DcVoltage	   			: REAL;
	r_DcCurrent				: REAL;
	r_DcPower				: REAL;

	Events					: ST_ACDCCharger_events;	

END_STRUCT
END_TYPE

// ---- POUs/Objects/ACDCCharger/Structs/ST_ACDCCharger_params.TcDUT
TYPE ST_ACDCCharger_params :
STRUCT
	b_ACDCChargerFitted		:	BOOL;
	ui_NrOfInstalledModules	:	UINT	:=	2;
	ui_ModuleDesignPower	:	Uint	:=	30;
	r_VoltageWindow			:	REAL	:=  2;
	GridVoltageHysteresis	: 	REAL	:=	2;
	BMSChargeLimitRampRate	:	REAL	:=	0.5; //DC amps per cycle;
	SocHysteresis			:	Real	:=	2;
END_STRUCT
END_TYPE

// ---- POUs/Objects/ACDCCharger/Structs/ST_ACDCCharger_set.TcDUT
TYPE ST_ACDCCharger_set :
STRUCT
	b_enable			: 	BOOL;
	e_ControlType		: 	ePowerControlType;
	r_currentSetpoint 	: 	REAL;
	r_powersetpoint		: 	REAL;
	r_MinGridVoltage	:	REAL;
	r_SocTarget			:	REAL;
END_STRUCT
END_TYPE

// ---- POUs/Objects/ACDCCharger/Structs/ST_SystemDiagnostic.TcDUT
TYPE ST_SystemDiagnostic :
STRUCT

    (* ===== GLOBAL STATUS ===== *)
    bAnyError          : BOOL;
    bAnyWarning        : BOOL;

    (* ===== ERRORS (CRITICAL) ===== *)
    bError_OutputOV    : BOOL;
    bError_OverTemp    : BOOL;
    bError_ShortCircuit: BOOL;
    bError_ModuleError : BOOL;
    bError_CommLost    : BOOL;
    bError_PhaseLost   : BOOL;

    (* ===== WARNINGS ===== *)
    bWarn_InputOV      : BOOL;
    bWarn_InputUV      : BOOL;
    bWarn_FanError     : BOOL;
    bWarn_PowerLimit   : BOOL;
    bWarn_TempHigh     : BOOL;
    bWarn_CurrentLimit : BOOL;

    (* ===== SYSTEM INFO ===== *)
    bAllModulesOff     : BOOL;
    bAllModulesOn      : BOOL;

END_STRUCT
END_TYPE

// ---- POUs/Objects/ACDCCharger/Structs/ST_SystemEval.TcDUT
TYPE ST_SystemEval :
STRUCT
    bAllModulesOff : BOOL;
    bAnyModuleActive : BOOL;
    bAnyModuleFault : BOOL;
    bGridOk : BOOL;

    rTotalAvailableCurrent : REAL;
    rMaxTemperature : REAL;
    iHealthyModules : INT;
END_STRUCT
END_TYPE

// ---- POUs/Objects/BMS/eNums/eBMS_Status.TcDUT
{attribute 'qualified_only'}
{attribute 'strict'}
{attribute 'to_string'} 
TYPE eBMS_Status :
(
	Init := 0,
	Normal := 1,
	FullCharge := 2,
	FullDischarge := 3,
	Warning := 4,
	Fault := 5,
	off := 6
);
END_TYPE

// ---- POUs/Objects/BMS/eNums/eHVDC_Powerstatus.TcDUT
{attribute 'qualified_only'}
{attribute 'strict'}
TYPE eHVDC_Powerstatus :
(
	OFF := 0,
	Precharging := 1,
	ON	:= 2	
);
END_TYPE

// ---- POUs/Objects/BMS/eNums/ePOUState.TcDUT
{attribute 'qualified_only'}
{attribute 'strict'}
TYPE ePOUState :
(
	OFF := 0,
	PowerUp := 1,
	Init := 2,
	Normal	:=	3,
	EMSTOP	:=	4,
	Shutdown := 5
);
END_TYPE

// ---- POUs/Objects/BMS/eNums/ePowerControl.TcDUT
{attribute 'qualified_only'}
{attribute 'strict'}
TYPE ePowerControl :
(
	Init := 0,
	Stay := 1,
	PowerOn := 2,
	PowerOff := 3
)word;
END_TYPE

// ---- POUs/Objects/BMS/eNums/ePowerOnStatus.TcDUT
{attribute 'qualified_only'}
{attribute 'strict'}
TYPE ePowerOnStatus :
(
	Off := 0,
	On	:= 1,
	PowerOn_Fault := 2,
	PowerOff_Fault := 3
)UINT;
END_TYPE

// ---- POUs/Objects/BMS/Structs/st_BMS_Events.TcDUT
TYPE st_BMS_Events :
STRUCT
	//sunspec error list
	b_COMMUNICATION_ERROR			:	BOOL;
	b_OVER_TEMP_ALARM				:	BOOL;
	b_OVER_TEMP_WARNING				:	BOOL;
	b_UNDER_TEMP_ALARM				:	BOOL;
	b_UNDER_TEMP_WARNING			:	BOOL;
	b_OVER_CHARGE_CURRENT_ALARM		:	BOOL;
	b_OVER_CHARGE_CURRENT_WARNING	:	BOOL;
	b_OVER_DISCHARGE_CURRENT_ALARM	:	BOOL;
	b_OVER_DISCHARGE_CURRENT_WARNING:	BOOL;
	b_OVER_VOLT_ALARM				:	BOOL;
	b_OVER_VOLT_WARNING				:	BOOL;
	b_UNDER_VOLT_ALARM				:	BOOL;
	b_UNDER_VOLT_WARNING			:	BOOL;
	b_UNDER_SOC_MIN_ALARM			:	BOOL;
	b_UNDER_SOC_MIN_WARNING			:	BOOL;
	b_OVER_SOC_MAX_ALARM			:	BOOL;
	b_OVER_SOC_MAX_WARNING			:	BOOL;
	b_VOLTAGE_IMBALANCE_WARNING		:	BOOL;
	b_TEMPERATURE_IMBALANCE_ALARM	:	BOOL;
	b_TEMPERATURE_IMBALANCE_WARNING	:	BOOL;
	b_CONTACTOR_ERROR				:	BOOL;
	b_FAN_ERROR						:	BOOL;
	b_GROUND_FAULT					:	BOOL;
	b_OPEN_DOOR_ERROR				:	BOOL;
	b_CURRENT_IMBALANCE_WARNING		:	BOOL;
	b_OTHER_ALARM					:	BOOL;
	b_OTHER_WARNING					:	BOOL;
	b_CONFIGURATION_ALARM			:	BOOL;
	b_CONFIGURATION_WARNING			:	BOOL;
	b_POWERONFAULT					: 	BOOL;
	b_POWEROFFFAULT					:	BOOL;
	b_DISCONNECTOR_OFF				: 	BOOL;
	b_MisingStrings					:	BOOL;
	
	b_SocLowLimitOutOfRange			:	BOOL;
	b_SocHighLimitOutOfRange		: 	BOOL;
	
	b_SBMUCommError					:	ARRAY [0..3] OF BOOL;	
	b_SBMUFailedToConnect			:	ARRAY [0..3] OF BOOL;
END_STRUCT
END_TYPE

// ---- POUs/Objects/BMS/Structs/st_BMS_Get.TcDUT
TYPE st_BMS_Get :
STRUCT
	BatteryInfo							: st_BMS_BatterySummary;
	
	T_RemainingTimeToAutoCalibration	: TIME;
	

	//detailed info	
	MBMU								:	st_MBMU_Status;
	SBMU								:	ARRAY[0..3] OF st_SBMU_Status;
	
	Events								:	st_BMS_Events;
END_STRUCT
END_TYPE

// ---- POUs/Objects/BMS/Structs/st_BMS_Params.TcDUT
TYPE st_BMS_Params :
STRUCT
	IP_BMS							:	STRING(16) := '192.168.1.60';
	r_SocHysteresis					:   REAL := 1; // % 
	r_SoCAbsoluteMin				: 	REAL := 6; // unscaled value
	r_SoCAbsoluteMax				: 	REAL := 100; //unscaled value

	r_KwhperString					: REAL := 208; //
	r_CrateBattery					: REAL := 0.5; //C
	r_AhperString					: REAL := 306; //Ah	
	b_DisableSOCAlarm				: BOOL := FALSE;
	b_ResetPersistentVars			: BOOL := FALSE;
	b_forcePrecharging				: BOOL := FALSE;
	r_InternalConditioningSoCMin	: REAL :=	10;
	
	T_AutoCalibrationInterval		: TIME := T#14D;
	b_EnableAutoCalibration			: BOOL := TRUE;
END_STRUCT
END_TYPE

// ---- POUs/Objects/BMS/Structs/st_BMS_BatterySummary.TcDUT
TYPE st_BMS_BatterySummary EXTENDS st_MBMU_BatterySummary :
STRUCT
	r_ratedPower				: REAL;
	r_ratedCurrent				: REAL;
	r_ratedEnergyCapacity		: REAL;
	ui_CycleCount				: UINT;
	r_SOCScaled					: REAL;
	b_chargingAllowed			: BOOL;
	b_dischargingAllowed		: BOOL;
	r_RemainingDischargeEnergyNett: REAL;
	r_RemainingChargeEnergyNett	: REAL;
	r_maxVoltageEver	 		: REAL;
	r_maxChargeCurrentEver		: REAL;
	r_maxDischargeCurrentEver	: REAL;
END_STRUCT
END_TYPE

// ---- POUs/Objects/BMS/Structs/st_BMS_Set.TcDUT
TYPE st_BMS_Set :
STRUCT
	b_enable	: BOOL := TRUE;
	r_SocMax	: REAL := 90;
	r_SocMin	: REAL := 10;
END_STRUCT
END_TYPE

// ---- POUs/Objects/BMS/Structs/st_MBMU_BatterySummary.TcDUT
TYPE st_MBMU_BatterySummary :
STRUCT
		//general
	b_BMSHeartBeatOK				:	BOOL;
	e_BMS_PowerOnStatus				:	ePowerOnStatus;
	e_BMS_Status					:	eBMS_Status;		

	r_SystemVoltage					:	REAL;
	r_SystemCurrent					:	REAL;
	r_SOC							:	REAL;
	r_SOH							:	REAL := 100;
	ar_CellVoltage					:	ARRAY[0..2] OF REAL;
	ar_CellTemperature				:	ARRAY[0..2] OF REAL;
	r_MaxChargeCurrentAllowed		:	REAL;
	r_MaxDischargeCurrentAllowed	:	REAL;
	r_MaxChargePowerAllowed			:	REAL;
	r_MaxDischargePowerAllowed		:	REAL;
	r_MaxSystemVoltageAllowed		:	REAL;
	r_MinSystemVoltageAllowed		:	REAL;
	
	r_SystemPower					:	REAL;
	r_ChargeSOE						:	REAL;
	r_DischargeSOE					:	REAL;
	
	r_RemainingChargeEnergy			:	REAL;
	r_RemainingDischargeEnergy		:	REAL;
	
	r_HistAccChargeEnergy			:	REAL;
	r_HistAccDischargeEnergy		:	REAL;
END_STRUCT	
END_TYPE

// ---- POUs/Objects/BMS/Structs/st_MBMU_Status.TcDUT
TYPE st_MBMU_Status :
STRUCT
	GeneralSBMUStatus			:	ARRAY [0..15] OF WORD;
	MBMUStatus					:	ARRAY [0..15] OF WORD;

	s_MBMU_SWVer				:	STRING(16);
	s_MBMU_HWVer				:	STRING(16);
	
	s_ETH_SWVer					:	STRING(32);
	r_ETH_HWVer					:	STRING(32);	
	
	by_NumberOfSubSystems		:	BYTE;
	DateTime					:	ARRAY[0..5] OF WORD;
	b_InsulationSwitchOpen		:	BOOL;
	
	BatteryStatus				:	st_MBMU_BatterySummary;
END_STRUCT
END_TYPE

// ---- POUs/Objects/BMS/Structs/st_SBMU_BatterySummary.TcDUT
TYPE st_SBMU_BatterySummary :
STRUCT
	r_SystemVoltage			:	REAL;
	r_SystemCurrent			:	REAL;
	r_SOC					:	REAL;
	r_SOH					:	REAL;
	ar_CellVoltage				:	ARRAY[0..2] OF REAL;
	ar_CellTemperature			:	ARRAY[0..2] OF REAL;
	r_MaxChargeCurrentAllowed		:	REAL;
	r_MaxDischargeCurrentAllowed	:	REAL;
	r_HistAccChargeEnergy			:	REAL;
	r_HistAccDischargeEnergy		:	REAL;
	
	//Gaan we hier uberhaupt iets mee doen?
	w_MaxVoltageCellLocation 	: 	WORD;//ARRAY[0..1] OF BYTE;
	w_MinVoltageCellLocation 	:	 WORD;//ARRAY[0..1] OF BYTE;
	w_MaxTempCellLocation 		: 	WORD;//ARRAY[0..1] OF BYTE;
	w_MinTempCellLocation 		: 	WORD;//ARRAY[0..1] OF BYTE;
END_STRUCT
END_TYPE

// ---- POUs/Objects/BMS/Structs/st_SBMU_Status.TcDUT
TYPE st_SBMU_Status :
STRUCT
	w_SystemWarning			:	WORD;
	SystemAlarm				:	ARRAY [0..2] OF WORD;
	
	b_PrechargeRelayClosed	:	BOOL;
	b_MainPosRelayClosed	:	BOOL;
	b_MainNegRelayClosed	:	BOOL;
	b_ControlBoxFanOn		:	BOOL;
	b_BalanceStatus			:	BOOL;
	b_DoorState				:	BOOL;	
	
	s_SBMU_SWVer			:	STRING(16);
	s_SBMU_HWVer			:	STRING(16);
	s_CSC_SWVer				:	STRING(16);
	s_CSC_HWVer				:	STRING(16);
	
	BatteryStatus			:	st_SBMU_BatterySummary;
END_STRUCT
END_TYPE

// ---- POUs/Objects/CoolingSystem/HeatpumpSystem/eNums/eHeatPumpMode.TcDUT
{attribute 'qualified_only'}
{attribute 'strict'}
{attribute 'to_string'}
TYPE eHeatPumpMode :
(
	Standby := 0,
	Cooling := 1,
	Heating := 2
)UINT := Standby;
END_TYPE

// ---- POUs/Objects/CoolingSystem/HeatpumpSystem/eNums/eHeatPumpState.TcDUT
{attribute 'qualified_only'}
{attribute 'strict'}
{attribute 'to_string'}
TYPE eHeatPumpState :
(
	OFF := 0,
	Initializing := 1,
	Standby := 2,
	Active_Cooling := 3,
	Active_Heating := 4,
	ERROR := 5
)UINT := OFF;
END_TYPE

// ---- POUs/Objects/CoolingSystem/HeatpumpSystem/eNums/eSupportedHeatpumps.TcDUT
{attribute 'qualified_only'}
{attribute 'strict'}
TYPE eSupportedHeatpumps :
(
	TranePicco := 0,
	LgThermaV	:= 1
);
END_TYPE

// ---- POUs/Objects/CoolingSystem/HeatpumpSystem/Structs/LG_Coils.TcDUT
TYPE LG_Coils :
STRUCT
	b_EnableOperation			:	BOOL := FALSE;
	b_EnableSwwOperation		: 	BOOL := FALSE;
	b_EnableSilentMode			:	BOOL := FALSE;
	b_EnableDesinfectionMode	:	BOOL := FALSE;
	b_EmstopActive				:	BOOL := FALSE;
	b_EnableEmStop				:	BOOL := FALSE;
END_STRUCT
END_TYPE

// ---- POUs/Objects/CoolingSystem/HeatpumpSystem/Structs/LG_ControlRegs.TcDUT
TYPE LG_ControlRegs :
STRUCT
	ui_OperatingMode	:	UINT := 3;
	ui_ControlMode		:	UINT := 1;
	r_Setpoint1			:	REAL := 20;
	r_RoomSetpoint		:	REAL;
	ui_TempShiftValue	:	UINT;
	r_setpoint2			:	REAL;
	r_RoomSetpoint2		:	REAL;
	ui_TempShiftValue2	:	UINT;
	r_DHWgoalTemp		:	REAL;
	ui_EnergyStatus		:	UINT := 2;	
END_STRUCT
END_TYPE

// ---- POUs/Objects/CoolingSystem/HeatpumpSystem/Structs/LG_get.TcDUT
TYPE LG_get :
STRUCT
	Coils	:	LG_Coils;
	Status	:	LG_StatusBits;
	Data	:	LG_InputRegs;
	Control	:	LG_ControlRegs;	
END_STRUCT
END_TYPE

// ---- POUs/Objects/CoolingSystem/HeatpumpSystem/Structs/LG_InputRegs.TcDUT
TYPE LG_InputRegs :
STRUCT
	UI_ErrorCode		:	UINT;
	ui_OperationalMode	:	UINT;
	r_CoolantInletTemp	:	REAL;
	r_CoolantOutletTemp	:	REAL;
	r_BackupHeaterTemp	:	REAL;
	r_SWWTankTemp		:	REAL;
	r_SolarCollectorTemp:	REAL;
	r_RoomTemp1			:	REAL;
	r_FlowRate			:	REAL;
	r_FlowTempCircuit2	:	REAL;
	r_RoomTemp2			:	REAL;
	UI_EnergyStatus		:	UINT;
	r_OutsideTemp		:	REAL;		
END_STRUCT
END_TYPE

// ---- POUs/Objects/CoolingSystem/HeatpumpSystem/Structs/LG_set.TcDUT
TYPE LG_set :
STRUCT
	Coils	:	LG_Coils;
	Regs	:	LG_ControlRegs;
END_STRUCT
END_TYPE

// ---- POUs/Objects/CoolingSystem/HeatpumpSystem/Structs/LG_Statusbits.TcDUT
TYPE LG_Statusbits :
STRUCT
	b_WaterFlowNOK				:	BOOL;
	b_WaterPumpOn				:	BOOL;
	b_ExtWaterPumpOn			:	BOOL;
	b_CompressorOn				:	BOOL;
	b_DefrostOn					:	BOOL;
	b_SWWModeOn					:	BOOL;
	b_SWWTankDesinfectionActive	:	BOOL;
	b_SilentModeOn				:	BOOL;
	b_CoolingActive				:	BOOL;
	b_SolarPumpActive			:	BOOL;
	b_BackupHeater1Active		:	BOOL;
	b_BackupHeater2Active		:	BOOL;
	b_SWWBoostHeaterActive		:	BOOL;
	b_ErrorActive				:	BOOL;
	b_EMOperationAvailable		:	BOOL;
	b_EMSWWOperationAvailable	:	BOOL;
	b_MixPumpActive				:	BOOL;
	
END_STRUCT
END_TYPE

// ---- POUs/Objects/CoolingSystem/HeatpumpSystem/Structs/ST_HeatpumpData.TcDUT
TYPE ST_HeatpumpData :
STRUCT
	i_FW_Version		:	INT;		//1
	i_FW_release		:	INT;		//2
	w_FW_Subrelease		:	WORD;		//3
	w_FW_creationDate	:	WORD;		//4
	
	w_Serialnumber		:	ARRAY[0..17] OF WORD;	//80-97
	
	i_OperatingHours	:	INT;		//305-317?
	
	r_CoolantPower		:  	REAL;
	r_InletWaterTemp	:	REAL;		//400
	r_OutletWaterTemp	:	REAL;		//401
	r_HighPressure		:	REAL;		//406
	r_LowPressure		:	REAL;		//414
	r_CompInputTemp		:	REAL;		//422
	r_OutdoorTemp		:	REAL;		//428
	r_CompOutputTemp	:	REAL;		//433-435
	ui_WaterFlowRate		:	UINT;		//444
	
	w_ErrorList			:	ARRAY[1..7] OF WORD;	//950-956	
	
	r_FanSpeedPCT		:	REAL;		//7000
	r_PumpSpeedPCT		:	REAL;		//7001
	
	r_SetpointHeating	:	REAL;		//7204
	r_SetpointCooling	:	REAL;		//7203
	b_DefrostingActive	:	BOOL;		//7214.14
END_STRUCT
END_TYPE

// ---- POUs/Objects/CoolingSystem/HeatpumpSystem/Structs/ST_HeatPumpEvents.TcDUT
TYPE ST_HeatPumpEvents :
STRUCT
	b_CommWarning		: BOOL;
	b_ProbeError		: BOOL;
	b_PressureError		: BOOL;
	b_CompressorError	: BOOL;
	b_ValveError		: BOOL;
	b_FanError			: BOOL;
	b_PumpError			: BOOL;
	b_WaterTempError	: BOOL;
	b_IOError			: BOOL;
	b_HeatpumpPreheatingActive	:	BOOL;
	b_TooColdForHeatpumpHeating	:	Bool;
END_STRUCT
END_TYPE

// ---- POUs/Objects/CoolingSystem/HeatpumpSystem/Structs/ST_HeatPump_Get.TcDUT
TYPE ST_HeatPump_Get :
STRUCT
	HeatPumpState 	: 	eHeatPumpState;
	Setpoint		:	REAL;
	Events			: 	ST_HeatPumpEvents;
	
	HeatpumpData	:	ST_HeatpumpData;
END_STRUCT
END_TYPE

// ---- POUs/Objects/CoolingSystem/HeatpumpSystem/Structs/ST_HeatPumpSystemEvents.TcDUT
TYPE ST_HeatPumpSystemEvents :
STRUCT

END_STRUCT
END_TYPE

// ---- POUs/Objects/CoolingSystem/HeatpumpSystem/Structs/ST_HeatpumpSystemGet.TcDUT
TYPE ST_HeatpumpSystemGet :
STRUCT
	HeatPumpStatus 			: 	eHeatPumpState;
	PrimaryHeatpumpGet		:	REFERENCE TO ST_HeatPump_Get;
	SecondaryHeatpumpGet 	:	REFERENCE TO ST_HeatPump_Get;
	//Heatpumps		:	REFERENCE TO ARRAY[1..2] OF ST_HeatPumpGet;
END_STRUCT
END_TYPE

// ---- POUs/Objects/CoolingSystem/HeatpumpSystem/Structs/st_OperatingPoint.TcDUT
TYPE st_OperatingPoint :
STRUCT
	OperatingMode	:	eHeatpumpMode;
	Setpoint		:	REAL;
END_STRUCT
END_TYPE

// ---- POUs/Objects/CoolingSystem/_Enum/eConditioningRequirement.TcDUT
{attribute 'qualified_only'}
{attribute 'strict'}
TYPE eConditioningRequirement :
(
	None := 0,
	Cooling := -1,
	Heating := +1
) int := None;
END_TYPE

// ---- POUs/Objects/CoolingSystem/_Enum/eCoolingSystemState.TcDUT
{attribute 'qualified_only'}
{attribute 'strict'}
{attribute 'to_string'}
TYPE eCoolingSystemState :
(
	OFF 						:= 	0,
	EnclosureConditioning 		:= 	1,
	InverterStartup 			:= 	2,
	BatteryConditioning 		:= 	3,
	InverterPowerMode 			:= 	5,
	DeHum						:= 	4,
	DehumEnding					:= 	6,
	InverterConditioning		:=  7,
	EMSTOP						:=	10
)uint := OFF;
END_TYPE

// ---- POUs/Objects/CoolingSystem/_Enum/ePumpState.TcDUT
{attribute 'qualified_only'}
{attribute 'strict'}
TYPE ePumpState :
(
	Off := 0,
	Starting := 1,
	Running	:= 2,
	Stopping := 3
);
END_TYPE

// ---- POUs/Objects/CoolingSystem/_Structs/ST_ConditioningRequirements.TcDUT
TYPE ST_ConditioningRequirements :
STRUCT
	//by_PSCoolingPowerMode	:	BYTE;
	//by_SetCooling			:	BYTE;
	Enclosure				:	eConditioningRequirement := 0;
	Battery					:	eConditioningRequirement := 0;
	Dehum					:	BOOL;
END_STRUCT
END_TYPE

// ---- POUs/Objects/CoolingSystem/_Structs/ST_CoolingSystem_Control.TcDUT
TYPE ST_CoolingSystem_Control :
STRUCT
	//system outputs
	b_CloseBatteryLoopValve		:	BOOL;
	b_CloseInverterLoopValve	:	BOOL;
	b_CloseFancoilLoopValve 	:	BOOL;
	
	b_BatteryLoopEnabled		:	BOOL;
	b_InverterLoopEnabled		:	BOOL;
	b_FancoilLoopEnabled		:	BOOL;
	
	b_DCFancoilEnable			: 	BOOL;
	b_DCPumpEnable 				: 	BOOL;
	b_ACPumpEnable				: 	BOOL;
	
	//System inputs
	r_EnclosureHumidity			:	REAL;
	r_EnclosureTemperature		:	REAL;
	r_CoolantTemperature		:	REAL;
	r_CoolantPressure			:	REAL;
	r_CoolantIdlePressure		:	REAL;
	
	r_CurrentEnclosureDewPoint	: 	REAL;
	
	//Inputs via main sequence
	//From BMS
	r_BMSBatteryTemperature		:	REAL;
	R_BMSMaxBatteryTemperature	: 	REAL;
	
	//From PowerModule
	b_InverterRunning			: 	BOOL;
	b_FanPowerstackEnable		:	BOOL;
	
	//HeatpumpData
	r_HeatPumpSetpoint			:	REAL;
	e_HeatpumpMode				:	eHeatPumpMode;
	HeatPumpStatus				:	eHeatPumpState;
	
	//From Internal power supply
	b_24V_Available				:	BOOL; 
	b_400v_Available			:	BOOL;
	e_400vSupplySource			: 	e400vSupplySource;
END_STRUCT
END_TYPE

// ---- POUs/Objects/CoolingSystem/_Structs/ST_CoolingSystem_Events.TcDUT
TYPE ST_CoolingSystem_Events :
STRUCT
	b_SystemOvertemperatureWarning	:	BOOL;
	b_SystemUnderTemperatureWarning :	BOOL;
	
	//faults
	b_CoolingSystemFuseFailure		: 	BOOL;
	b_ACwaterPumpTimeOut			: 	BOOL;	
	
	b_InverterLoopValveStuck		: 	BOOL;
	b_BattLoopValveStuck			: 	BOOL;
	b_FancoilLoopValveStuck			: 	BOOL;

	b_DCpumpPressureFault			: 	BOOL;
	b_DCpumpTimeout					:	BOOL;
	
	//System pressure dropped below idle minimum pressure. suspect coolant loss.
	b_CoolingLoopIdlePressureWarning 	: 	BOOL := FALSE;	
	b_CoolingLoopIdlePressureError 		: 	BOOL := FALSE;	
	
	//Systempressure too low during conditioning, possible pump failure or coolant loss.
	b_InverterCoolingLoopError 		: 	BOOL := FALSE;

	b_HeatpumpWarning				:	BOOL;
	b_HeatPumpError					: 	BOOL;
	
	//Temperature errors
	b_CoolantTempTooLow				: 	BOOL;
	b_CoolantTempLow				: 	BOOL;
	b_CoolantTempTooHigh			: 	BOOL;
	b_CoolantTempHigh				: 	BOOL;
END_STRUCT
END_TYPE

// ---- POUs/Objects/CoolingSystem/_Structs/ST_CoolingSystem_Get.TcDUT
TYPE ST_CoolingSystem_Get :
STRUCT
	CoolingSystemMode		:	eCoolingSystemState;
	HeatPumpStatus			: 	eHeatPumpState;
	r_CoolantTemperature	:	REAL;
	r_CoolantPressure		:	REAL;
	r_EnclosureDewpoint		:	REAL;
	ui_DehumRemainingTime	: 	UINT; //minutes
		
	
	HeatPumpSystem 			: REFERENCE TO ST_HeatpumpSystemGet;	
	Events					: ST_CoolingSystem_Events;
END_STRUCT
END_TYPE

// ---- POUs/Objects/CoolingSystem/_Structs/ST_CoolingSystem_Inputs.TcDUT
TYPE ST_CoolingSystem_Inputs :
STRUCT
	BattLoopValveFB					:	BOOL;
	InvLoopValveFB					:	BOOL;
	FancoilLoopValveFB				:	BOOL;
	
	CoolingLoopPressureSensor 		:	INT;
	CoolingLoopTemperatureSensor 	:	INT;
	
	CoolingSystem400VFuseFB			:	BOOL;
	ACPumpFb						: 	BOOL;
	
END_STRUCT
END_TYPE

// ---- POUs/Objects/CoolingSystem/_Structs/ST_CoolingSystem_Outputs.TcDUT
TYPE ST_CoolingSystem_Outputs :
STRUCT
	DCFanEnable						:	BOOL;
	
	BattLoopValveClose				:	BOOL;
	InvLoopValveClose				:	BOOL;
	FancoilLoopValveClose			:	BOOL;
		
	DCPumpEnable					: 	BOOL;
	ACPumpEnable					: 	BOOL;
END_STRUCT
END_TYPE

// ---- POUs/Objects/CoolingSystem/_Structs/ST_Coolingsystem_params.TcDUT
TYPE ST_Coolingsystem_params :
STRUCT
	b_ActivateCooling						: BOOL;
	b_ActivateHeating						: BOOL;	
	
	r_MaxInverterTemperature				: REAL := 50;

	r_MaxCoolantTemperature					: REAL := 40;
	r_CoolantTempCoolingStart				: REAL := 35;
	r_CoolantTempHeatingStart				: REAL := 0;
	r_MinCoolantTemperature					: REAL := -20;

	r_EnclosureIdleTempMin					: REAL := 10.0;
	r_EnclosureIdleTempMax					: REAL := 40.0;
	
	r_BatteryTempMin						: REAL := 15.0;
	r_BatteryTempHysteresis					: REAL := 5;
	r_BatteryTempMax						: REAL := 40.0;
	b_DoubleHeatpump						: BOOL := FALSE;
	
	// Minimum base coolant pressure
	r_MinimumSystemBasePressureWarningLevel	: REAL := 1;
	r_MinimumSystemBasePressureErrorLevel	: REAL := 0.7;
	r_PressureHysteresis					: REAL := 0.2;
	// Minimum cooling system pressure increase with 24V pump running
	r_StartupPumpMinimumPressure			: REAL	:= 0.1;
	// minimum cooling system pressure increase with main pump running
	r_MainPumpMinimumPressure				: REAL	:= 0.2;
	b_MainPumpFbInstalled					: BOOL := FALSE;
	
	//Allowed pressure drop during stable operation, measured against a 5 minutes average pressure
	AllowedCoolantPressureDrop				:	REAL := 0.25;
	
	i_MaximumValveOperatingTime				: INT := 10; //in s
	
	i_modbusRetries								: INT := 30;
	t_ModbusTimeout								:	TIME := T#2S;
	PrimaryHeatpumpAddr							:	BYTE := 1;
	HeatpumpType							: 	eSupportedHeatpumps := eSupportedHeatpumps.LgThermaV;
	LGCoilSettings								:	BYTE := 2#0000_0001;
	SecondaryHeatpumpAddr						:	BYTE := 2;
	dw_HeatpumpOperationDelay					: DWORD := 30; // minutes
	
	//If the heatpump has run within this timeframe, no preheating is required before operation can start
	i_SkipHPPreheatingTime						: 	INT		:= 60; //minutes. 
	r_MinimumCoolantTemperatureForHPHeatingMode	:	REAL	:= 15;
END_STRUCT
END_TYPE

// ---- POUs/Objects/CoolingSystem/_Enum/eCoolingControl.TcDUT
{attribute 'qualified_only'}
{attribute 'strict'}
TYPE eCoolingControl :
(
	off := 0,
	temporary := 1,
	full := 2
);
END_TYPE

// ---- POUs/Objects/CoolingSystem/_Enum/eCoolingPowerRequest.TcDUT
{attribute 'qualified_only'}
{attribute 'strict'}
TYPE eCoolingPowerRequest :
(
	off := 0,
	intern := 1,
	full := 2
);
END_TYPE

// ---- POUs/Objects/DCSwitchgear/ST_DCSwitchgear_Get.TcDUT
TYPE ST_DCSwitchgear_Get :
STRUCT
	b_CouplingState					: BOOL;
	r_Current						: REAL;
	r_Power							: REAL;
	r_Voltage						: REAL;
	r_RatedCurrent					: REAL;
END_STRUCT
END_TYPE

// ---- POUs/Objects/Enclosure/Climate/ST_Enclosureclimate_events.TcDUT
TYPE ST_Enclosureclimate_events :
STRUCT
	b_HumidityHigh 			: BOOL;
	b_HumidityTooHigh 		: BOOL;
	b_TemperatureHigh		: BOOL;
	b_TemperatureTooHigh	: BOOL;
	b_TemperatureLow		: BOOL;
	b_TemperatureTooLow		: BOOL;
	b_AIOverrange			: BOOL;
	b_AIUnderrange			: BOOL;
	b_AIError				: BOOL;
	b_DewpointTooHigh		: BOOL;
END_STRUCT
END_TYPE

// ---- POUs/Objects/Enclosure/Climate/ST_EnclosureClimate_get.TcDUT
TYPE ST_EnclosureClimate_get :
STRUCT
	r_Humidity			: REAL;
	r_Temperature		: REAL;
	
	events				: ST_EnclosureClimate_events;
END_STRUCT
END_TYPE

// ---- POUs/Objects/Enclosure/Climate/ST_EnclosureClimate_Params.TcDUT
TYPE ST_EnclosureClimate_Params :
STRUCT
	r_HumidityHysteris		: REAL:= 2;
	r_HumidityHigh			: REAL:= 80;
	r_HumidityTooHigh		: REAL:= 90;
	r_TemperatureHysteris	: REAL:= 2;
	r_TemperatureHigh		: REAL:= 40;
	r_TemperatureTooHigh	: REAL:= 50;
	r_TemperatureLow		: REAL:= -10;
	r_TemperatureTooLow		: REAL:= -20;
END_STRUCT
END_TYPE

// ---- POUs/Objects/Enclosure/Doors/ST_DoorsNLocks_get.TcDUT
TYPE ST_DoorsNLocks_get :
STRUCT
	b_ClientpanelDoorClosed			: BOOL;
	b_ControlPanelDoorClosed		: BOOL;	
END_STRUCT
END_TYPE

// ---- POUs/Objects/Enclosure/LedIndicator/BeckhoffController/eDCstate.TcDUT
{attribute 'qualified_only'}
{attribute 'strict'}
TYPE eDCstate :
(
	charging :=-1,
	idle := 0,
	discharging := 1
);
END_TYPE

// ---- POUs/Objects/Enclosure/LedIndicator/BeckhoffController/eLEDSteps.TcDUT
{attribute 'qualified_only'}
{attribute 'strict'}
TYPE eLEDSteps :
(
	initialise,	
	running
);
END_TYPE

// ---- POUs/Objects/Enclosure/LedIndicator/BeckhoffController/LEDColor.TcDUT
TYPE LEDColor :
STRUCT	
	red 	:USINT;
	green	:USINT;
	blue	:USINT;
	white	:USINT;
END_STRUCT
END_TYPE

// ---- POUs/Objects/Enclosure/LedIndicator/BeckhoffController/LEDCommands.TcDUT
TYPE LEDCommands :
STRUCT
	
	fill 		: USINT := 1;
	clear 		: USINT	:= 2;
	copy 		: USINT	:= 3;
	movePixel 	: USINT	:= 4;
	reverse 	: USINT	:= 7;
END_STRUCT
END_TYPE

// ---- POUs/Objects/Enclosure/LedIndicator/BeckhoffController/LEDControl.TcDUT
TYPE LEDControl :
STRUCT
	execute 	: BIT;
	send		: BIT;
	update		: BIT;
	command		: USINT;(*LEDCommands*)
	index 		: UINT;
	length		: UINT;
	parameter	: UINT;
	color 		: LEDColor;
END_STRUCT
END_TYPE

// ---- POUs/Objects/Enclosure/LedIndicator/BeckhoffController/LEDStatus.TcDUT
TYPE LEDStatus :
STRUCT
	busy				: BIT;
	transmit			: BIT;
	sendAcknowledge 	: BIT;
	updateAcknowledge	: BIT;
	commandAcknowledge	: BIT;
	commandReject		: BIT;
	warning				: BIT;
	error				: BIT;
	InputCycleCounter	: USINT;
END_STRUCT
END_TYPE

// ---- POUs/Objects/Enclosure/LedIndicator/BeckhoffController/eSystemStatus.TcDUT
{attribute 'qualified_only'}
{attribute 'strict'}
TYPE eSystemStatus :
(
	off			:= 0,	// off
	neutral 	:= 1, 	(*white*)
	normal		:= 2, 	// green
	attention	:= 3,	// blue 100charge 0discharge
	warning		:= 4,	// yellow
	error		:= 5	// red	
) BYTE;
END_TYPE

// ---- POUs/Objects/Enclosure/LedIndicator/eColorOrder.TcDUT
{attribute 'qualified_only'}

TYPE eColorOrder :
(
	RGB := 0,
	GRB := 1
);
END_TYPE

// ---- POUs/Objects/Enclosure/LedIndicator/ST_Ledstrip_get.TcDUT
TYPE ST_Ledstrip_get :
STRUCT
	b_error		: BOOL;
	BeckhoffLed	: BOOL;
END_STRUCT
END_TYPE

// ---- POUs/Objects/Enclosure/LedIndicator/st_Ledstrip_MachineData.TcDUT
TYPE st_Ledstrip_MachineData :
STRUCT
	r_SOC 					: REAL;
	r_DCCurrent				: REAL;
	e_systemStatus 			: eSystemStatus;
END_STRUCT
END_TYPE

// ---- POUs/Objects/Enclosure/LedIndicator/st_Ledstrip_params.TcDUT
TYPE st_Ledstrip_params :
STRUCT
	IP				: STRING 	:= '192.168.1.43'; //arduino controller only
	Numleds			: BYTE		:= 116;
	ColorOrder		: eColorOrder := eColorOrder.GRB;
END_STRUCT
END_TYPE

// ---- POUs/Objects/Enclosure/_struct/ST_Enclosure_get.TcDUT
TYPE ST_Enclosure_get :
STRUCT
	climate				: ST_EnclosureClimate_Get;
	doors				: ST_DoorsNLocks_get;
	ledstrip			: ST_Ledstrip_get;
END_STRUCT
END_TYPE

// ---- POUs/Objects/Enclosure/_struct/st_Enclosure_params.TcDUT
TYPE st_Enclosure_params :
STRUCT
	climate			: ST_EnclosureClimate_params;
	ledstrip		: st_Ledstrip_params;
END_STRUCT
END_TYPE

// ---- POUs/Objects/Enclosure/_struct/ST_enclosure_set.TcDUT
TYPE ST_enclosure_set :
STRUCT
	by_LedBrightness 	: BYTE := 100;
END_STRUCT
END_TYPE

// ---- POUs/Objects/GenComm/eNums/eGenControlProtocol.TcDUT
{attribute 'qualified_only'}
{attribute 'strict'}
TYPE eGenControlProtocol :
(
	None := 0,
	AGC150 := 1
);
END_TYPE

// ---- POUs/Objects/GenComm/eNums/eGenOperationMode.TcDUT
{attribute 'qualified_only'}
{attribute 'strict'}
TYPE eGenOperationMode :
(
	None := 0,
	BlockMode := 1,
	ManualMode := 2,
	SemiAuto := 3,
	Auto	:=	4,
	Test	:=	5
);
END_TYPE

// ---- POUs/Objects/GenComm/eNums/eOnOffState.TcDUT
{attribute 'qualified_only'}
{attribute 'strict'}
TYPE eOnOffState :
(
	none := 0,
	Enable := 1,
	Disable := 2
);
END_TYPE

// ---- POUs/Objects/GenComm/Structs/ST_Genset_Get.TcDUT
TYPE ST_Genset_Get :
STRUCT
	CommunicationOK		: 	BOOL;
	FuelLow				: 	BOOL;
	FuelCritical		: 	BOOL;
		
	bGenBreakerClosed	:	BOOL;
	bMainBreakerClosed	:	BOOL;
	bGenRunning			:	BOOL;
	bGenVoltFreqOK		:	BOOL;
	bMainsFailure		:	BOOL;
	
	eActiveGenMode		:	eGenOperationMode;
	bIslandModeActive	:	BOOL;
	bAMFActive			:	BOOL;
	bPeakshaveActive	:	BOOL;
	bFixedPowerActive	:	BOOL;

	ar_LineVoltage	:	ARRAY[0..3] OF REAL;
	ar_PhaseVoltage	:	ARRAY[0..3] OF REAL;
	ar_Frequency	:	ARRAY[0..3] OF REAL;
	ar_Current		:	ARRAY[0..3] OF REAL;
	ar_PowerFactor	: 	ARRAY[0..0] OF REAL;
	ar_ActivePower 	:   ARRAY[0..3] OF REAL;
	ar_ReactivePower: 	ARRAY[0..0] OF REAL;
	ar_ApparentPower:	ARRAY[0..0] OF REAL;
	
	
END_STRUCT
END_TYPE

// ---- POUs/Objects/GenComm/Structs/ST_AGC150_Set.TcDUT
TYPE ST_AGC150_Set :
STRUCT
	IP					:	STRING	:=	'192.168.2.21';
	DroopEnable			: 	BOOL;
	GenOn				:	eOnOffState := eOnOffState.none;
	GenBreakerOn		:	eOnOffState := eOnOffState.none;	
	MainBreakerON		:	eOnOffState := eOnOffState.none;
	GenAutoSyncOn		:	eOnOffState := eOnOffState.none;
	OperationMode		:	eGenOperationMode := eGenOperationMode.Auto;
	AutoStartStop		:	BOOL;
	
	bIslandModeEnable		:	BOOL;
	bAMFModeEnable			:	BOOL;
	bPeakshavingEnable		: 	BOOL;
	bFixedPowerEnable		:	BOOL := TRUE;
	bMPE					:	BOOL;

	Pset			:	REAL;	//0..100%
	Qset			:	REAL;	//60..100 = 0.6..1
	PFset			:	REAL := 1;	//-100..100%
	FreqRegulator	:	REAL; 	//-100..100 = -10..+10% of nominal
	VoltRegulator	:	REAL; 	//-100..100 = -10..+10% of nominal
	U_Fdroopset		: 	REAL := 4; 	//0..100 = 0..+10% of nominal
END_STRUCT
END_TYPE

// ---- POUs/Objects/GenComm/Structs/ST_GenComm_Params.TcDUT
TYPE ST_GenComm_Params :
STRUCT
	IP					:	STRING	:=	'192.168.2.21';
	GenControlProtocol	: 	eGenControlProtocol := eGenControlProtocol.None;
END_STRUCT
END_TYPE

// ---- POUs/Objects/GenComm/Structs/ST_Genset_Set.TcDUT
TYPE ST_Genset_Set :
STRUCT
	enable			:  	BOOL;
	StartStop		:	BOOL; //true = start;
	Pset			:	REAL;	//0..100%
	Qset			:	REAL;	//60..100 = 0.6..1
	PFset			:	REAL;	//0 - 1;
	Uset			: 	REAL;
	Fset			: 	REAL;
	U_Fdroopset		: 	REAL := 4;
	GensetMode		: 	eGensetMode := eGensetMode.FixedPower;
END_STRUCT
END_TYPE

// ---- POUs/Objects/HartingIO/ST_HartingIO_get.TcDUT
TYPE ST_HartingIO_get :
STRUCT
	b_DigitalInput1Active		:	BOOL;
	b_DigitalInput2Active		:	BOOL;
	b_GenLowFuel				:	BOOL;
	b_ExtSystemShutdownRequest	:	BOOL;
	b_ExtEMstopOK				: 	BOOL;
	b_ExtEMstopActive			: 	BOOL;
END_STRUCT
END_TYPE

// ---- POUs/Objects/HartingIO/ST_HartingIO_params.TcDUT
TYPE ST_HartingIO_params :
STRUCT
	PrimaryOutputContactSignal		: 	eOutputContactSignal := eOutputContactSignal.GenStartStop;
	SecondaryOutputContactSignal	:	eOutputContactSignal := eOutputContactSignal.None;
	PrimaryInputContactSignal		: 	eInputSignal := eInputSignal.None;
	SecondaryInputContactSignal		: 	eInputSignal := eInputSignal.None;
	AO1Target				: eAOTarget := eAOTarget.Genset;
	AO2Target				: eAOTarget	:= eAOTarget.hPU;
END_STRUCT
END_TYPE

// ---- POUs/Objects/HartingIO/ST_HartingIO_set.TcDUT
TYPE ST_HartingIO_set :
STRUCT
	w_SwitchControlSignals		: 	WORD; // control signals for output contact
	r_manualAnalogOutput		: 	REAL; // 0 - 100%
	r_gensetAnalogOutput		: 	REAL; // 0 - 100%
	r_HpuAnalogOutput			: 	REAL; // 0 - 100%
END_STRUCT
END_TYPE

// ---- POUs/Objects/HartingIO/_Enum/eAOTarget.TcDUT
{attribute 'qualified_only'}
{attribute 'strict'}
TYPE eAOTarget:
(
	manual 	:= 0,
	Genset	:= 1,
	hPU		:= 2
);
END_TYPE

// ---- POUs/Objects/HartingIO/_Enum/eOutputContactSignal.TcDUT
{attribute 'qualified_only'}

TYPE eOutputContactSignal :
(
	None 			:= 	0,
	FireAlarm 		:= 	1,
	GenStartStop 	:= 	2,
	HPU				:= 	3,
	SystemActive	:=	4,
	PVenable		:= 	5,
	ManualOpen		:=	99,
	ManualClose		:=	100
) UINT;
END_TYPE

// ---- POUs/Objects/HartingIO/_Enum/eInputSignal.TcDUT
{attribute 'qualified_only'}

TYPE eInputSignal :
(
	None 			:= 	0,
	GenLowFuel 		:= 	1,
	StopOperation 	:= 	2,
	EMstop			:=	3
) UINT;
END_TYPE

// ---- POUs/Objects/InterMachineCom/ST_InterMachineCom_Master.TcDUT
TYPE ST_InterMachineCom_Master :
STRUCT
	PS		: REAL; //Power setpoint, scale 0.1% 
	QS		: REAL; // Reactive Setpoint, scale 0.1%
	CW		: WORD; // ControlWord, b0: Start, b1: Stop, b2: shutdown, b3: EMstop, b4: Reset, b15: watchdog signal
END_STRUCT
END_TYPE

// ---- POUs/Objects/InterMachineCom/ST_IntermachineCom_params.TcDUT
TYPE ST_IntermachineCom_params :
STRUCT
	InternalBrokerIP		: STRING := '10.4.0.41';
	MasterPublishRate		: TIME := T#20MS;
	SlavePublishRate		: TIME := T#1S;
	WatchdogPulseRate		: TIME := T#2S;
	EMstopCoupling			: BOOL;
END_STRUCT
END_TYPE

// ---- POUs/Objects/InterMachineCom/st_InterMachineCom_Slave.TcDUT
TYPE st_InterMachineCom_Slave :
STRUCT
	ACP : UINT; //available charge power [kW]
	ADP	: UINT; //available discharge power [kW]
	AQ	: UINT; //available Reactive Power [kvar]
	SW	: WORD; //status word: b0: standby, b1: running, b2: Stopped, b3: Discharge Only, b4: Charge Only, b5: warning active, b6: Alarm active, b7: EMstop active, b15: watchdogbit
END_STRUCT
END_TYPE

// ---- POUs/Objects/InterMachineCom/ST_InterMachineCom_SlaveConData.TcDUT
TYPE ST_InterMachineCom_SlaveConData :
STRUCT
	enable			: BOOL;
	BrokerIP		: STRING;
END_STRUCT
END_TYPE

// ---- POUs/Objects/InternalPowerSupply/eNums/e400VSupplySource.TcDUT
{attribute 'qualified_only'}
{attribute 'strict'}
{attribute 'to_string'}

TYPE e400VSupplySource :
(
	none := 0,
	grid := 1,
	CEE := 2
);
END_TYPE

// ---- POUs/Objects/InternalPowerSupply/eNums/eSupplyState.TcDUT
{attribute 'qualified_only'}
{attribute 'strict'}
TYPE eSupplyState :
(
	enum_member := 0
);
END_TYPE

// ---- POUs/Objects/InternalPowerSupply/Structs/ST_InternalPowerStatus.TcDUT
TYPE ST_InternalPowerStatus :
STRUCT
	b_Status_24VDC		:	BOOL;
	b_Status_HVDC		:	BOOL;
	b_Status_400VAC		:	BOOL;
END_STRUCT
END_TYPE

// ---- POUs/Objects/InternalPowerSupply/Structs/ST_InternalPowerSupply_Events.TcDUT
TYPE ST_InternalPowerSupply_Events :
STRUCT
	b_DCPSUFault				: 	BOOL; //fuse blown or psu_ok signal lost
	b_ACPSUFault				: 	BOOL;
	b_GridInputFuseTripped		:	BOOL;
	b_CEEInputFuseTripped		:	BOOL;
	b_HVDCShutdownTimeExceeded	:	BOOL;
	b_UPSLowShutdown			:	BOOL;	//System shutdown event when ups battery drains during operation
END_STRUCT
END_TYPE

// ---- POUs/Objects/InternalPowerSupply/Structs/ST_InternalPowerSupply_Get.TcDUT
TYPE ST_InternalPowerSupply_Get :
STRUCT
	b_24VdcAvailable	:	BOOL;
	b_HVDCAvailable		:	BOOL;
	b_400VACAvailable	:	BOOL;	
	e_400VSupplySource	: 	e400VSupplySource;
	
	UPS					:	REFERENCE TO ST_UPSGet;	
	Events				:	st_InternalPowerSupply_Events;
END_STRUCT
END_TYPE

// ---- POUs/Objects/InternalPowerSupply/Structs/ST_InternalPowerSupply_Params.TcDUT
TYPE ST_InternalPowerSupply_Params :
STRUCT
	b_InternalACfromBusbar	: BOOL := FALSE;
	i_IntZPTStartupDelay: INT := 100; // ms
	i_ACStartupDelay : INT := 100; //ms
	i_DCPSU_StartupDelay: INT := 5000; //ms
	i_ACPSU_StartupDelay: INT := 5000; //ms
	
	//trigger level before Battery low error is issued. 
	usi_UPSBattLowErrorSOC		:	USINT 	:= 30;
	//UPS charging request was apparently denied. System should shutdown? 
	usi_UPSBattLowwarningSOC	:	USINT 	:= 40;
	//trigger level before Battery low warning is issued and UPS charging is requested from Internal power supply
	usi_UPSBattLowinfoSOC		:	USINT	:= 60;	
	//r_SOC level at which UPS charging is no longer requested so HVDC can be shutdown.
	usi_UPSBattOKSOC 			:	USINT	:= 90;
	//Timeout between LowBatteryError occuring and self-shutdown initiating
	LowBatteryShutdownTimer		:	TIME := T#10M;
END_STRUCT
END_TYPE

// ---- POUs/Objects/InternalPowerSupply/Structs/ST_InternalPowerSupply_PowerDemand.TcDUT
TYPE ST_InternalPowerSupply_PowerDemand :
STRUCT
	b_Demand_24V	:	BOOL;
	b_Demand_400V	:	BOOL;
	b_Demand_HVDC	:	BOOL;
END_STRUCT
END_TYPE

// ---- POUs/Objects/InternalPowerSupply/UPS/eNums/eUPSState.TcDUT
{attribute 'qualified_only'}
{attribute 'strict'}
TYPE eUPSState :
(
	Inoperative 	:= 0,
	Input_Active	:= 1,
	On_Battery		:= 2
);
END_TYPE

// ---- POUs/Objects/InternalPowerSupply/UPS/Structs/ST_UPSData.TcDUT
TYPE ST_UPSData :
STRUCT
	udi_StatusFunctions 		: 	UDINT;
	udi_StatusInterface 		: 	UDINT;
	ui_InputVoltage				:	UINT;
	ui_InputCurrent				:	UINT;
	ui_OutputVoltage			:	UINT;
	ui_OutputCurrent			:	UINT;
	ui_BatteryVoltage			: 	UINT;
	ui_BatteryChargingCurrent 	: 	UINT;
	ui_BatteryTemperature 		: 	UINT;
	ui_DeviceTemperature		: 	UINT;
	udi_SOC 					:	UDINT;
	ui_TuPCShutdown				:	UINT;
	ui_SOH						:	UINT;
END_STRUCT
END_TYPE

// ---- POUs/Objects/InternalPowerSupply/UPS/Structs/ST_UPSEvents.TcDUT
TYPE ST_UPSEvents :
STRUCT
	b_BatteryLowInfo		:	BOOL;	//initialize DC conditioning
	b_BatteryLowWarning		:	BOOL;	//Battery charging failed, consider shutdown
	b_BatteryLowError		:	BOOL;	//Battery level critical, System should shutdown
	b_NoBatteryError		:	BOOL;	//no Battery voltage detected?
	b_InputVoltageWarning	:	BOOL;	//ipsstate says 24v is available, but no input is seen.
END_STRUCT
END_TYPE

// ---- POUs/Objects/InternalPowerSupply/UPS/Structs/ST_UPSGET.TcDUT
TYPE ST_UPSGET :
STRUCT
	r_InputVoltage		:	REAL;
	r_OutputVoltage		:	REAL;
	r_BatteryVoltage	:	REAL;
	r_OutputCurrent		: 	REAL;
	ui_SOC				:	UINT	:=	100;
	
	b_ChargerActive		:	BOOL;
	b_SystemOnBattery	:	BOOL;
	b_SystemOnDCInput		:	BOOL;
	
	Events			:	ST_UPSEvents;
END_STRUCT
END_TYPE

// ---- POUs/Objects/NeutralTransformer/_Struct/ST_NeutralTransformer_events.TcDUT
TYPE ST_NeutralTransformer_events :
STRUCT
	b_TemperatureHighPhase						: ARRAY [1..3] OF BOOL; //1=L1, 2=L2, 3=L3
	b_TemperatureTooHighPhase					: ARRAY [1..3] OF BOOL; //1=L1, 2=L2, 3=L3
	b_VoltageUnbalanceHigh										: BOOL;
	b_VoltageUnbalanceTooHigh									: BOOL;
	b_NeutralCurrentHigh										: BOOL;
	b_NeutralCurrentTooHigh										: BOOL;
	
	b_OvercurrentWarning										: BOOL;
	b_OvercurrentAlarm											: BOOL;
END_STRUCT
END_TYPE

// ---- POUs/Objects/NeutralTransformer/_Struct/ST_NeutralTransformer_Get.TcDUT
TYPE ST_NeutralTransformer_Get :
STRUCT
	b_active									: BOOL;
	r_TemperaturePhase							: ARRAY [0..6] OF REAL;
	r_Powerload									: REAL;
	r_ratedPower								: REAL; //kva
	events										: ST_NeutralTransformer_events;
END_STRUCT
END_TYPE

// ---- POUs/Objects/NeutralTransformer/_Struct/ST_Neutraltransformer_params.TcDUT
TYPE ST_Neutraltransformer_params :
STRUCT
	ui_ratedpower					: UINT := 60; // kVA
	by_TemperatureHighWarning		: BYTE := 80;
	by_TemperatureHighAlarm			: BYTE := 90;
	ui_TemperatureHighTripDelay		: UINT := 10; // seconds
	by_VoltageUnbalanceWarning		: BYTE := 10; // %
	by_VoltageUnbalanceAlarm		: BYTE := 20; // %
	ui_VoltageUnbalanceTripDelay	: UINT := 10;// seconds
	r_OCTripFactor					: REAL := 1.4;  //Overcurrent trip factor software
END_STRUCT
END_TYPE

// ---- POUs/Objects/PeakshaveBox/DUTs/ePsbCtRange.TcDUT
{attribute 'qualified_only'}
TYPE ePsbCtRange :
(
	_100A := 100,
	_250A := 250,
	_400A := 400,
	_630A := 630,
	_1000A := 1000,
	_1500A := 1500,
	_2000A := 2000,
	_4000A := 4000
) UINT := _1000A;
END_TYPE

// ---- POUs/Objects/PeakshaveBox/DUTs/ePSBMode.TcDUT
{attribute 'qualified_only'}
{attribute 'strict'}
{attribute 'to_string'}
TYPE ePSBMode :
(
	None 				:= 0,
	Monitor				:= 1,
	MonitorControl		:= 2	
);
END_TYPE

// ---- POUs/Objects/PeakshaveBox/DUTs/ePSBhardware.TcDUT
{attribute 'qualified_only'}
TYPE ePSBhardware :
(
	Wago := 0,
	Beckhoff := 1
); 
END_TYPE

// ---- POUs/Objects/PeakshaveBox/DUTs/ST_PowerMeasurement_status.TcDUT
TYPE ST_PowerMeasurement_status :
STRUCT
	b_RotaryField	: BOOL;
	b_GeneralWarning: BOOL;
	b_GeneralFault	: BOOL;
	b_OverVoltage 	: BOOL;
	b_UnderVoltage	: BOOL;
	b_OverCurrent	: BOOL;
	b_Error_Phase 	: ARRAY [1..3] OF BOOL;
END_STRUCT
END_TYPE

// ---- POUs/Objects/PeakshaveBox/ST_peakshavebox_params.TcDUT
TYPE ST_peakshavebox_params :
STRUCT
	PSBhardware			: ePSBhardware := ePSBHardware.Beckhoff; // if enabled, psb v2 is configured.
	fastmode 			: BOOL := TRUE; // only in old PSB
END_STRUCT
END_TYPE

// ---- POUs/Objects/PeakshaveBox/ST_PeakshaveBox_Set.TcDUT
TYPE ST_PeakshaveBox_Set :
STRUCT
	b_ContactorClose : BOOL;
	b_Alarm			 : BOOL;
	b_ExtIO			 : BOOL;
	b_BreakerControl : BOOL;
	ui_CtRange		 : UINT := 1000;
	r_VTRatio		 : REAL := 1;
	b_InverseCTdirection: BOOL;
END_STRUCT
END_TYPE

// ---- POUs/Objects/PLCStatus/Enum/eFTPState.TcDUT
{attribute 'qualified_only'}
{attribute 'strict'}
{attribute 'to_string'}
TYPE
	eFTPState :(
		Disconnected := 0,	
		Connecting := 1,      
		Downloading := 2,      
		Success := 3,    
		Failure := 4
	);
END_TYPE

// ---- POUs/Objects/PLCStatus/Enum/eNetcomState.TcDUT
{attribute 'qualified_only'}
{attribute 'strict'}
{attribute 'To_string'}
TYPE eNetcomState :
(
	NotConnected := 0,
	OK:=1,
	Warning:=2,
	Error:=3
);
END_TYPE

// ---- POUs/Objects/PLCStatus/Enum/eInstalState.TcDUT
{attribute 'qualified_only'}
{attribute 'strict'}
TYPE eInstalState :
(
	InProgress := 0,
	Success	   := 1,
	Failure	   := 2
);
END_TYPE

// ---- POUs/Objects/PLCStatus/ST_EL9410.TcDUT
TYPE ST_EL9410 :
STRUCT
	bit_UpUndervoltage	: BIT;
	bit_UsUndervoltage	: BIT;
	ui_state			: UINT;
END_STRUCT
END_TYPE

// ---- POUs/Objects/PLCStatus/ST_PLCstate_get.TcDUT
TYPE ST_PLCstate_get :
STRUCT
	r_CPUload		: REAL;
	e_ProfinetState	: eNetcomState;
	e_EthercatState	: eNetcomState;
END_STRUCT
END_TYPE

// ---- POUs/Objects/PLCStatus/ST_PLC_events.TcDUT
TYPE ST_PLC_events :
STRUCT
	b_EthercatMasterFault		: BOOL;
END_STRUCT
END_TYPE

// ---- POUs/Objects/PowerQualityMonitor/_Enums/eACRotationState.TcDUT
{attribute 'qualified_only'}
{attribute 'strict'}
{attribute 'to_string'}
TYPE eACRotationState :
(
	Left := -1,
	None := 0,
	Right := 1
);
END_TYPE

// ---- POUs/Objects/PowerQualityMonitor/_Structs/ST_MeasurementFieldData.TcDUT
TYPE ST_MeasurementFieldData :
STRUCT
	//Power
	ar_ApparentPower			: 	ARRAY[0..3] OF REAL;
	ar_ReactivePower			: 	ARRAY[0..3] OF REAL;
	ar_ActivePower				: 	ARRAY[0..3] OF REAL;

	//Energy Consumed
	r_EnergyConsumed			:	REAL := 0;
	
	//Energy Delivered
	r_EnergySupplied			:	REAL := 0;
	
	//THD
	ar_THD						:	ARRAY[0..3] OF REAL := [0, 0, 0, 0];	
	
	//PF
	ar_PowerFactor				:	ARRAY[0..3] OF REAL := [0, 0, 0, 0];
	
	//Current
	ar_Current					: 	ARRAY[0..4] OF REAL := [0, 0, 0, 0];
	r_CurrentUnbalance			:	REAL;
END_STRUCT
END_TYPE

// ---- POUs/Objects/PowerQualityMonitor/_Structs/ST_MeasurementVoltageData.TcDUT
TYPE ST_MeasurementVoltageData EXTENDS ST_MeasurementFieldData:
STRUCT
	e_ACrotationStatus		:	eACRotationState;
	ar_PhaseVoltage			: 	ARRAY[0..3] OF REAL;
	ar_LineVoltage			:	ARRAY[0..3] OF REAL;
	li_TimeVoltZeroCrossup 	: 	LINT;
	ar_Frequency			: 	ARRAY[0..3] OF REAL;
	r_VoltageUnbalance		: 	REAL;	
END_STRUCT
END_TYPE

// ---- POUs/Objects/PowerQualityMonitor/_Structs/ST_PowerMonitor_BESS.TcDUT
TYPE ST_PowerMonitor_BESS :
STRUCT
	e_ACrotationStatus			: 	eACrotationState;
	ar_Current					:	ARRAY [0..4] OF REAL;
	r_LineVoltage				: 	REAL;
	r_Frequency					: 	REAL;
	r_currentUnbalance			:	REAL;
	//Power
	r_ApparentPower				: 	REAL;
	r_ReactivePower				: 	REAL;
	r_ActivePower				: 	REAL;
	//Energy Consumed
	r_EnergyConsumed			:	REAL;
	
	//Energy Delivered
	r_EnergySupplied			:	REAL;
	
	r_PowerFactor 				:	REAL;
END_STRUCT
END_TYPE

// ---- POUs/Objects/PowerQualityMonitor/_Structs/ST_PowerMonitor_Events.TcDUT
TYPE ST_PowerMonitor_Events :
STRUCT
	b_MBCommWarning 		: BOOL;
	b_MBCommError 			: BOOL;
	b_MBTimeoutWarning 		: BOOL;
	b_EL3443Warning			: BOOL;
	b_EL3443Error		: BOOL;
	b_ACdirectionDataInvalid: BOOL;
END_STRUCT
END_TYPE

// ---- POUs/Objects/PowerQualityMonitor/_Structs/ST_PowerMonitor_get.TcDUT
TYPE ST_PowerMonitor_get :
STRUCT
	PQMeterReady		: 	BOOL;
	InputField			:	ST_PowerMonitor_InputField;	
	OutputField			:	ST_PowerMonitor_OutputField;
	InternalSupply 		: 	ST_MeasurementFieldData;
	
	//Inverter power/energy input & output
	BESS				:	ST_PowerMonitor_BESS;
	events				:	ST_PowerMonitor_Events;
END_STRUCT
END_TYPE

// ---- POUs/Objects/PowerQualityMonitor/_Structs/ST_PowerMonitor_InputField.TcDUT
TYPE ST_PowerMonitor_InputField EXTENDS st_MeasurementVoltageData:
STRUCT
	r_loadshare			: 	REAL;
	Powerlock			: 	ARRAY [1..2] OF ST_MeasurementFieldData;
END_STRUCT
END_TYPE

// ---- POUs/Objects/PowerQualityMonitor/_Structs/ST_PowerMonitor_OutputField.TcDUT
TYPE ST_PowerMonitor_OutputField EXTENDS st_MeasurementVoltageData:
STRUCT
	r_loadshare					: 	REAL;
	Powerlock					: 	ARRAY [1..3] OF ST_MeasurementFieldData;
END_STRUCT
END_TYPE

// ---- POUs/Objects/PowerStack/NetContactor/eNetcontMode.TcDUT
{attribute 'qualified_only'}
{attribute 'strict'}
TYPE eNetcontMode :
(
	auto := 0,
	left := 1,
	right := 2,
	none := 3
);
END_TYPE

// ---- POUs/Objects/PowerStack/NetContactor/_Structs/ST_Netcontactor_Events.TcDUT
TYPE ST_Netcontactor_Events :
STRUCT
	b_AMFEnabled							: BOOL;
	b_ContactorRightFbFault					: BOOL;
	b_ContactorLeftFbFault					: BOOL;
	b_ContactorFbTimeout					: BOOL;
	b_PhaseRotationFault					: BOOL;
	b_IllegalLeftFieldSelected				: BOOL;
END_STRUCT
END_TYPE

// ---- POUs/Objects/PowerStack/NetContactor/_Structs/ST_Netcontactor_get.TcDUT
TYPE ST_Netcontactor_get :
STRUCT
	e_NetConState					: eNetcontactorState;
	b_SyncCloseCommand				: BOOL;
	b_NetConFb						: BOOL;
	b_NetcontRightFb				: BOOL;
	b_NetcontLeftFb					: BOOL;
	events							: ST_Netcontactor_events;
END_STRUCT
END_TYPE

// ---- POUs/Objects/PowerStack/NetContactor/_Structs/ST_Netcontactor_set.TcDUT
TYPE ST_Netcontactor_set :
STRUCT
	e_ACRotationState				: eACRotationState; // 0:No AC, 1: AC CLOCKWISE, 2: AC ANTI-CLOCKWISE
	e_ClosingRequest				: eNetcontMode;
	b_ACdetected					: BOOL;
	b_RotationSwitchEnable			: BOOL;
	b_SynchronizedToD7				: BOOL;
END_STRUCT
END_TYPE

// ---- POUs/Objects/PowerStack/_Enums/eInverterModes.TcDUT
{attribute 'qualified_only'}
{attribute 'strict'}
{attribute 'to_string'}
TYPE eInverterModes :
(
	Afe := 0,
	Island := 1,
	Microgrid := 2
);
END_TYPE

// ---- POUs/Objects/PowerStack/_Enums/eNetContactorState.TcDUT
{attribute 'qualified_only'}
{attribute 'strict'}
{attribute 'to_string'}
TYPE eNetContactorState :
(
	Open 			:= 0,
	RightClosed		:= 1,
	LeftClosed		:= 2
);
END_TYPE

// ---- POUs/Objects/PowerStack/_Enums/ePowerModes.TcDUT
{attribute 'qualified_only'}
{attribute 'strict'}
{attribute 'to_string'}
TYPE ePowerModes :
(
	DroopZeroStart 		:= 0,
	Droop				:= 1,
	Isochronous			:= 2
);
END_TYPE

// ---- POUs/Objects/PowerStack/_Enums/ePowerModuleThrottlingState.TcDUT
{attribute 'qualified_only'}
{attribute 'strict'}
TYPE ePowerModuleThrottlingState :
(
	None := 0,
	FilterTemp := 1,
	InverterTemp:= 2,
	Overvoltage := 3
);
END_TYPE

// ---- POUs/Objects/PowerStack/_Enums/ePowerstate.TcDUT
{attribute 'qualified_only'}
{attribute 'strict'}
TYPE ePowerstate :
(
	Charging := -1,
	None := 0,
	Discharging := 1		
)INT;
END_TYPE

// ---- POUs/Objects/PowerStack/_Enums/eStatusPowerModule.TcDUT
{attribute 'qualified_only'}
{attribute 'strict'}
{attribute 'to_string'}
TYPE eStatusPowerModule :
(
	Init					:= 0,	// Not ready to do anything yet
	off						:= 1, 	// OFF MCCBs OPEN,
	DcOK					:= 2, 	// Dc voltage above 80%
	idle					:= 3, 	// MCCB CLOSED, No modulation
	running					:= 4,	// MCCB CLOSED + Modulation	
	fault					:= 10,
	EMStop					:= 11
);
END_TYPE

// ---- POUs/Objects/PowerStack/_Enums/eStatusPowerStack.TcDUT
{attribute 'qualified_only'}
{attribute 'strict'}
{attribute 'to_string'}
TYPE eStatusPowerStack :
(
	Init					:= 0,	// Not ready to do anything yet
	off						:= 1, 	// OFF MCCBs OPEN,
	idle					:= 2, 	// MCCB CLOSED, No modulation, Netcontactor CLOSED with grid OR Netcontactor OPEN + modulation with no grid
	running					:= 3,	// MCCB CLOSED + Modulation, Netcontactor CLOSED
	ecorunning				:= 4,	// MCCB CLOSED + Modulation with only one out of two inverters, Netcontactor CLOSED
	Wait_CoolingMode1		:= 20,
	Wait_HVDC				:= 21,
	Start_Master			:= 22, 	// Starting master
	Start_Slave				:= 23,	// Starting slave
	Synchronization			:= 24,
	Wait_CoolingMode2		:= 25,
	Standby					:= 9,
	Standby_GridSupply		:= 10, 	// POWERMODULE 1 + 2 off, Netcontactor Closed
	Standby_InternalSupply	:= 11,	// PowerModule 1 ON, powermodule 2 Off, Netcontactor OPEN
	shutdown				:= 12,
	fault					:= 13,
	GridCodeStop			:= 14,
	Cooling_Shutdown		:= 15  // 	
);		
END_TYPE

// ---- POUs/Objects/PowerStack/_Enums/ePLM.TcDUT
{attribute 'qualified_only'}
{attribute 'strict'}
{attribute 'to_string'}

TYPE ePLM: //power limiting 
(
	FreqShift := 0,
	VoltShift := 1,
	FreqVoltShift := 2,
	Shutdown := 3
);
END_TYPE

// ---- POUs/Objects/PowerStack/_Structs/NestedStructs/ST_Powermodule_CalibData.TcDUT
TYPE ST_Powermodule_CalibData :
STRUCT
	Pset: ARRAY[0..4] OF REAL;
	Qset: ARRAY[0..4] OF REAL;
	Pmeas: ARRAY[0..4] OF ARRAY[0..4] OF REAL;
	Qmeas: ARRAY[0..4] OF ARRAY[0..4] OF REAL;
END_STRUCT
END_TYPE

// ---- POUs/Objects/PowerStack/_Structs/NestedStructs/ST_InverterControlWord.TcDUT
TYPE ST_InverterControlWord :
STRUCT
	b_ChargeDC				: BOOL;
	b_run					: BOOL;
	b_Reset					: BOOL;
	b_FieldbusControlEnable	: BOOL;
	b_WatchdogPulse			: BOOL;
	b_ParallelAFE			: BOOL;
	b_PIDenable				: BOOL;
	b_GridCodeEnable		: BOOL;
	b_ExtGridcodeTrip		: BOOL;
END_STRUCT
END_TYPE

// ---- POUs/Objects/PowerStack/_Structs/NestedStructs/ST_Inverter_StatusWord.TcDUT
TYPE ST_Inverter_StatusWord :
STRUCT
	//General Status Word Variables
		b_ReadyToDCCharge				: BOOL;
		b_ReadyToOperate				: BOOL;
		b_Running						: BOOL;
		b_Fault							: BOOL;
		b_RunEnabled					: BOOL;
		b_QuickstopNotActive			: BOOL;
		b_MCCBControlNotOK				: BOOL;
		b_Warning						: BOOL;
		b_DCAtReference					: BOOL;
		b_DCAboveLimit					: BOOL;
		b_WatchdogFeedback				: BOOL;
END_STRUCT
END_TYPE

// ---- POUs/Objects/PowerStack/_Structs/NestedStructs/ST_Inverter_UgridStatusWord.TcDUT
TYPE ST_Inverter_UgridStatusWord :
STRUCT
	//Ugrid Status Word
		b_ChargeControlActive			: BOOL;
		b_InternalChargingSwitchStatus	: BOOL;
		b_MCBcontrol					: BOOL;
		b_MCBStatus						: BOOL;
		b_RunEnabled					: BOOL;
		b_DriveReady					: BOOL;
		b_AFEmodeActive					: BOOL;
		b_IslandModeActive				: BOOL;
		b_MicrogridModeActive			: BOOL;
		b_RunRequestActive				: BOOL;
		b_DriveInRunState				: BOOL;
		b_FaultActive					: BOOL;
		b_SynchronizedToD7				: BOOL;
		b_D7MeasurementsOK				: BOOL;	
END_STRUCT
END_TYPE

// ---- POUs/Objects/PowerStack/_Structs/NestedStructs/ST_Inverter_additionalTemperatures.TcDUT
TYPE ST_Inverter_additionalTemperatures :
STRUCT
	r_ambient					: REAL;
	r_CMchokeOuter				: ARRAY[1..4] OF REAL;
	r_CMchokeInner				: ARRAY[1..4] OF REAL;
	r_GrChokeOuter				: ARRAY[1..3] OF REAL;
	r_GrChokeInner				: ARRAY[1..3] OF REAL;
	r_ACCapsTop					: REAL;
	r_ACCapsBottom				: REAL;
	r_DCCaps					: REAL;
	r_ACbusbarOutput			: REAL;
	r_ACbusbarCMchoke			: REAL;
	r_DCbusbarCMChoke			: REAL;
	r_AirInletModule			: REAL;
	r_AirOutletFancoil			: REAL;
	r_WaterInletFancoil			: REAL;
	r_WaterOutletFancoil		: REAL;
	r_FancoilCompartement		: REAL;
END_STRUCT
END_TYPE

// ---- POUs/Objects/PowerStack/_Structs/NestedStructs/ST_Inverter_LineState.TcDUT
TYPE ST_Inverter_LineState :
STRUCT
	b_LineVoltTripLimHigh		: BOOL;
	b_LineVoltTripLimlow		: BOOL;
	b_LineFreqTripLimHigh		: BOOL;
	b_LineFreqTripLimLow		: BOOL;
	b_LineFreqOK				: BOOL;
	b_LineVoltOK				: BOOL;
	b_FRTActive					: BOOL;
	b_GridCodeTripActive		: BOOL;
END_STRUCT
END_TYPE

// ---- POUs/Objects/PowerStack/_Structs/NestedStructs/ST_Inverter_Write.TcDUT
TYPE ST_Inverter_Write :
STRUCT
	Controlword				: ST_InverterControlWord;
	ui_ControlwordValue		: UINT;
	i_invertermode 			: INT;
	i_BaseCurrentRef 		: INT;
	i_ReactiveCurrentRef	: INT;
	i_FrequencyDroop		: INT;
	i_VoltageDroop			: INT;
	i_FrequencyDroopOffset	: INT;
	i_VoltageCorrection		: INT;
	i_BaseRefRampRate		: INT;
	i_StartPowerMode		: INT;
	i_StartVoltageMode		: INT;
	i_OutActCurrentLimit	: INT;
	i_InActCurrentLimit		: INT;
	i_DCVramprate			: INT;
END_STRUCT
END_TYPE

// ---- POUs/Objects/PowerStack/_Structs/NestedStructs/ST_Powermodule_Events.TcDUT
TYPE ST_Powermodule_Events :
STRUCT
		b_GeneralFaultFlag				: BOOL;
		b_GeneralWarningFlag			: BOOL;

		//Powermodule Warnings
		b_CMSTemperatureRangeWarning	: BOOL;
		b_FanStateUnknownWarning		: BOOL;
		b_TempThrottlingActive			: BOOL;
		b_CurrThrottlingActive			: BOOL;
		
		//INVERTER Fault Status Word 
		b_F1OverCurrent					: BOOL;
		b_F2OverVoltage					: BOOL;
		b_F9UnderVoltage				: BOOL;
		b_F91ShortCircuit				: BOOL;
		b_F3EarthFault					: BOOL;
		b_Spare							: BOOL;
		b_F14UnitOverTemperature		: BOOL;
		b_F56TemperatureFault			: BOOL;
		b_F10LineSynchFault				: BOOL;
		b_F52KeypadOCCommFault			: BOOL;
		b_F53FieldbusFault				: BOOL;
		b_F59SystembusFault				: BOOL;
		b_F54SlotCommunicationFault		: BOOL;
		b_F50Meas4mAFault				: BOOL;
		b_F11OutputPhaseFault 			: BOOL;
		b_F80ChargeFault				: BOOL;
		b_F51ExternalFault				: BOOL;
		b_F31IGBTFault					: BOOL;
		b_F64MCBstateFault				: BOOL;
		b_WatchdogError					: BOOL;
		b_24VdcUVRFault					: BOOL;
		
		//Buscoupler connected faults
		b_MCCBtrip						: BOOL;	
		b_ShutdownTimeOut				: BOOL;
		b_StartUpTimeOut				: BOOL;
	
		//Temperature faults and warnings 
		b_CMChokeTemperatureHigh		: ARRAY [1..4] OF BOOL;
		b_CMChokeTemperatureTooHigh		: ARRAY [1..4] OF BOOL;
		b_GridChokeTemperatureHigh		: ARRAY [1..3] OF BOOL;
		b_GridChokeTemperatureTooHigh	: ARRAY [1..3] OF BOOL;
		b_inverterTemperatureHigh		: BOOL;
		b_PT100Overrange				: BOOL;
		b_PT100Underrange				: BOOL;
		by_PT100ErrorCount				: BYTE;
		

		
END_STRUCT
END_TYPE

// ---- POUs/Objects/PowerStack/_Structs/NestedStructs/ST_Powermodule_PowerCurveCoefficients.TcDUT
TYPE ST_Powermodule_PowerCurveCoefficients :
STRUCT
	enable: BOOL;
	a : REAL;
	b : REAL;
	c : REAL;
	d : REAL; 
	e : REAL;
	f : REAL;
END_STRUCT
END_TYPE

// ---- POUs/Objects/PowerStack/_Structs/NestedStructs/ST_PowerStack_Events.TcDUT
TYPE ST_PowerStack_Events :
STRUCT
	//INFO
	b_CoolingDerating				: BOOL;
	b_PlimitShiftingActive			: BOOL;
	
	//Warnings
	b_DCdeviationHigh				: BOOL;
	b_TemperatureWarning			: BOOL;
	b_OvercurrentWarning			: BOOL;
	b_UndervoltageWarning			: BOOL;
	b_OvervoltageWarning			: BOOL;
	b_TemperatureDeviationHigh		: BOOL;
	b_PlimitShutdownWarning			: BOOL;
	
	b_MasterWarning					: BOOL;
	b_SlaveWarning					: BOOL;
	b_GridCodeWarning				: BOOL;
	
	//faults
	b_UnderFreqFault				: BOOL;
	b_OverFreqFault					: BOOL;
	b_UnderVoltageFault				: BOOL;
	b_OverVoltageFault				: BOOL;
	b_OvercurrentFault				: BOOL;
	b_PlimitShutdown				: BOOL;
	b_TemperatureFault				: BOOL;
	b_MasterFault					: BOOL;
	b_SlaveFault					: BOOL;
	b_NetcontactorFault				: BOOL;
	
	
	b_startupTimeOut				: BOOL;
	b_ShutdownTimeOut				: BOOL;
	
	ui_shutdownRemainingTime		: UINT;
END_STRUCT
END_TYPE

// ---- POUs/Objects/PowerStack/_Structs/NestedStructs/ST_Powerstack_ShiftingParams.TcDUT
TYPE ST_Powerstack_ShiftingParams :
STRUCT
	InitialOverloadDelay		: TIME := T#1S; // ignore initial power surge
	ShutdownDelay				: TIME := T#1M; // shutdown delay when limit is exceeded.
	ShiftingHoldTime			: TIME := T#20M; // when shifting is applied, this time must pass before returning back.
	ShiftingRate				: TIME := T#100MS; // time per step. Number of steps is + and - 1000. The stepsize is 1/2000 of the set min / max range.
	FreqMaxPu					: REAL := 1.03; //per unit
	FreqMinPu					: REAL := 0.97;
	VoltMaxPu					: REAL := 1.1;
	VoltMinPu					: REAL := 0.9;
END_STRUCT
END_TYPE

// ---- POUs/Objects/PowerStack/_Structs/ST_PowerModule_calibration.TcDUT
TYPE ST_PowerModule_calibration :
STRUCT
	b_StartCalibration			: BOOL;
	r_Pset						: REAL;
	r_Qset						: REAL;
	PCoefficients				: ST_Powermodule_PowerCurveCoefficients;
	QCoefficients				: ST_Powermodule_PowerCurveCoefficients;
	CalibrationData				: ST_Powermodule_calibData;
END_STRUCT
END_TYPE

// ---- POUs/Objects/PowerStack/_Structs/ST_PowerModule_params.TcDUT
TYPE ST_PowerModule_params :
STRUCT
	b_FieldBusControlEnable			: BOOL := TRUE;
	r_InverterRatedCurrent			: REAL := 460; //Ampere // according danfoss grid current rating
	r_InverterRatedPower			: REAL := 360; //kva // according rated max current
	r_tempfanOn						: REAL := 50;
	r_powerLoadFanOn				: REAL := 30;	
	r_ACCurrentLimitMax				: REAL := 650;
	r_ACcurrentLimitMin				: REAL := 100;
	r_FilterTempWarning				: REAL := 80; //also used for throttling start
	r_FilterTempAlarm				: REAL := 90; //also used for for throttling end 
	r_InverterTempWarning			: REAL := 55; //also used for throttling start
	r_InverterTempAlarm				: REAL := 60; //also used for for throttling end 
	i_VoltageOffset					: INT := 4; //correction factor voltage control.
	i_DCVramprate					: INT := 200;
	ui_DCVoltageDeltaPrechargeOK	: UINT := 20; // VDC
	ui_DCvoltageMinPrechargeOK		: UINT := 590; //VDC
	r_ModulationIndexLimit			: REAL := 98; 
	r_ModulationIndexLimitHyst		: REAL := 0.5; 
	r_ThrottlingMinimum				: REAL := 0.3;
END_STRUCT
END_TYPE

// ---- POUs/Objects/PowerStack/_Structs/ST_PowerModule_get.TcDUT
TYPE ST_PowerModule_get :
STRUCT
	b_online						: BOOL;

